LIN {X 0,Y 403.463,Z 460.03,A -85,B 0,C 180,E1 17685.281,E2 17685.281} C_VEL
LIN {X 0,Y 392.488,Z 442.787,A -85,B 0,C 180,E1 17683.008,E2 17683.008} C_VEL
LIN {X 0,Y 381.726,Z 427.301,A -85,B 0,C 180,E1 17680.568,E2 17680.568} C_VEL
LIN {X 0,Y 370.448,Z 412.508,A -85,B 0,C 180,E1 17677.735,E2 17677.735} C_VEL
LIN {X 0,Y 365.323,Z 406.384,A -85,B 0,C 180,E1 17676.338,E2 17676.338} C_VEL
LIN {X 0,Y 362.446,Z 402.418,A -85,B 0,C 180,E1 17675.403,E2 17675.403} C_VEL
LIN {X 0,Y 359.831,Z 397.717,A -85,B 0,C 180,E1 17673.762,E2 17673.762} C_VEL
LIN {X 0,Y 358.471,Z 395.72,A -85,B 0,C 180,E1 17672.95,E2 17672.95} C_VEL
LIN {X 0,Y 356.459,Z 391.629,A -85,B 0,C 180,E1 17671.448,E2 17671.448} C_VEL
LIN {X 0,Y 354.433,Z 388.786,A -85,B 0,C 180,E1 17670.142,E2 17670.142} C_VEL
LIN {X 0,Y 353.887,Z 386.869,A -85,B 0,C 180,E1 17669.398,E2 17669.398} C_VEL
LIN {X 0,Y 353.858,Z 386.651,A -85,B 0,C 180,E1 17665.436,E2 17665.436} C_VEL
LIN {X 0,Y 353.853,Z 386.657,A -85,B 0,C 180,E1 17661.204,E2 17661.204} C_VEL
LIN {X 0,Y 353.849,Z 386.658,A -85,B 0,C 180,E1 17657.09,E2 17657.09} C_VEL
LIN {X 0,Y 353.851,Z 386.655,A -85,B 0,C 180,E1 17653.065,E2 17653.065} C_VEL
LIN {X 0,Y 353.847,Z 386.65,A -85,B 0,C 180,E1 17648.941,E2 17648.941} C_VEL
LIN {X 0,Y 353.843,Z 386.642,A -85,B 0,C 180,E1 17644.863,E2 17644.863} C_VEL
LIN {X 0,Y 353.835,Z 386.641,A -85,B 0,C 180,E1 17640.648,E2 17640.648} C_VEL
LIN {X 0,Y 353.831,Z 386.639,A -85,B 0,C 180,E1 17636.598,E2 17636.598} C_VEL
LIN {X 0,Y 353.837,Z 386.638,A -85,B 0,C 180,E1 17632.532,E2 17632.532} C_VEL
LIN {X 0,Y 353.829,Z 386.639,A -85,B 0,C 180,E1 17628.426,E2 17628.426} C_VEL
LIN {X 0,Y 353.825,Z 386.642,A -85,B 0,C 180,E1 17624.26,E2 17624.26} C_VEL
LIN {X 0,Y 353.839,Z 386.746,A -85,B 0,C 180,E1 17620.523,E2 17620.523} C_VEL
LIN {X 0,Y 354.207,Z 388.34,A -85,B 0,C 180,E1 17619.856,E2 17619.856} C_VEL
LIN {X 0,Y 356.199,Z 391.406,A -85,B 0,C 180,E1 17618.598,E2 17618.598} C_VEL
LIN {X 0,Y 357.309,Z 392.844,A -85,B 0,C 180,E1 17617.978,E2 17617.978} C_VEL
LIN {X 0,Y 359.294,Z 396.484,A -85,B 0,C 180,E1 17616.724,E2 17616.724} C_VEL
LIN {X 0,Y 360.473,Z 398.042,A -85,B 0,C 180,E1 17616.111,E2 17616.111} C_VEL
LIN {X 0,Y 362.61,Z 401.899,A -85,B 0,C 180,E1 17614.873,E2 17614.873} C_VEL
LIN {X 0,Y 363.731,Z 403.854,A -85,B 0,C 180,E1 17614.258,E2 17614.258} C_VEL
LIN {X 0,Y 366.651,Z 408.927,A -85,B 0,C 180,E1 17612.734,E2 17612.734} C_VEL
LIN {X 0,Y 369.981,Z 414.917,A -85,B 0,C 180,E1 17611.07,E2 17611.07} C_VEL
LIN {X 0,Y 374.091,Z 422.477,A -85,B 0,C 180,E1 17609.125,E2 17609.125} C_VEL
LIN {X 0,Y 380.392,Z 434.798,A -85,B 0,C 180,E1 17606.316,E2 17606.316} C_VEL
LIN {X 0,Y 382.59,Z 438.943,A -85,B 0,C 180,E1 17605.52,E2 17605.52} C_VEL
LIN {X 0,Y 392.217,Z 454.061,A -85,B 0,C 180,E1 17603.311,E2 17603.311} C_VEL
LIN {X 0,Y 402.215,Z 471.066,A -85,B 0,C 180,E1 17601.19,E2 17601.19} C_VEL
LIN {X 0,Y 403.176,Z 473.296,A -85,B 0,C 180,E1 17600.98,E2 17600.98} C_VEL
LIN {X 0,Y 405.136,Z 498.631,A -85,B 0,C 180,E1 17600.003,E2 17600.003} C_VEL
LIN {X 0,Y 395.268,Z 723.239,A -85,B 0,C 180,E1 17595.557,E2 17595.557} C_VEL
LIN {X 0,Y 393.737,Z 748.587,A -85,B 0,C 180,E1 17594.972,E2 17594.972} C_VEL
LIN {X 0,Y 391.268,Z 771.267,A -85,B 0,C 180,E1 17594.239,E2 17594.239} C_VEL
LIN {X 0,Y 388.306,Z 792.146,A -85,B 0,C 180,E1 17593.329,E2 17593.329} C_VEL
LIN {X 0,Y 384.904,Z 812.358,A -85,B 0,C 180,E1 17592.178,E2 17592.178} C_VEL
LIN {X 0,Y 380.795,Z 834.172,A -85,B 0,C 180,E1 17590.626,E2 17590.626} C_VEL
LIN {X 0,Y 376.722,Z 854.159,A -85,B 0,C 180,E1 17588.876,E2 17588.876} C_VEL
LIN {X 0,Y 372.707,Z 872.71,A -85,B 0,C 180,E1 17586.924,E2 17586.924} C_VEL
LIN {X 0,Y 368.756,Z 890.411,A -85,B 0,C 180,E1 17584.705,E2 17584.705} C_VEL
LIN {X 0,Y 364.732,Z 908.565,A -85,B 0,C 180,E1 17582.013,E2 17582.013} C_VEL
LIN {X 0,Y 361.461,Z 924.026,A -85,B 0,C 180,E1 17579.312,E2 17579.312} C_VEL
LIN {X 0,Y 358.561,Z 938.566,A -85,B 0,C 180,E1 17576.317,E2 17576.317} C_VEL
LIN {X 0,Y 356.353,Z 950.961,A -85,B 0,C 180,E1 17573.303,E2 17573.303} C_VEL
LIN {X 0,Y 354.62,Z 962.641,A -85,B 0,C 180,E1 17569.946,E2 17569.946} C_VEL
LIN {X 0,Y 353.535,Z 972.315,A -85,B 0,C 180,E1 17566.596,E2 17566.596} C_VEL
LIN {X 0,Y 352.953,Z 979.977,A -85,B 0,C 180,E1 17563.264,E2 17563.264} C_VEL
LIN {X 0,Y 352.727,Z 985.943,A -85,B 0,C 180,E1 17559.957,E2 17559.957} C_VEL
LIN {X 0,Y 352.729,Z 989.818,A -85,B 0,C 180,E1 17557.001,E2 17557.001} C_VEL
LIN {X 0,Y 352.826,Z 992.572,A -85,B 0,C 180,E1 17553.737,E2 17553.737} C_VEL
LIN {X 0,Y 352.867,Z 993.592,A -85,B 0,C 180,E1 17550.812,E2 17550.812} C_VEL
LIN {X 0,Y 352.842,Z 993.283,A -85,B 0,C 180,E1 17547.727,E2 17547.727} C_VEL
LIN {X 0,Y 352.785,Z 991.52,A -85,B 0,C 180,E1 17544.798,E2 17544.798} C_VEL
LIN {X 0,Y 352.717,Z 988.222,A -85,B 0,C 180,E1 17541.616,E2 17541.616} C_VEL
LIN {X 0,Y 352.811,Z 983.168,A -85,B 0,C 180,E1 17538.394,E2 17538.394} C_VEL
LIN {X 0,Y 353.17,Z 976.363,A -85,B 0,C 180,E1 17535.073,E2 17535.073} C_VEL
LIN {X 0,Y 353.949,Z 968.18,A -85,B 0,C 180,E1 17531.899,E2 17531.899} C_VEL
LIN {X 0,Y 355.322,Z 957.64,A -85,B 0,C 180,E1 17528.545,E2 17528.545} C_VEL
LIN {X 0,Y 357.259,Z 945.699,A -85,B 0,C 180,E1 17525.358,E2 17525.358} C_VEL
LIN {X 0,Y 359.753,Z 932.382,A -85,B 0,C 180,E1 17522.349,E2 17522.349} C_VEL
LIN {X 0,Y 362.762,Z 917.65,A -85,B 0,C 180,E1 17519.53,E2 17519.53} C_VEL
LIN {X 0,Y 366.487,Z 900.583,A -85,B 0,C 180,E1 17516.749,E2 17516.749} C_VEL
LIN {X 0,Y 370.396,Z 883.117,A -85,B 0,C 180,E1 17514.338,E2 17514.338} C_VEL
LIN {X 0,Y 374.564,Z 864.11,A -85,B 0,C 180,E1 17512.129,E2 17512.129} C_VEL
LIN {X 0,Y 378.612,Z 844.945,A -85,B 0,C 180,E1 17510.282,E2 17510.282} C_VEL
LIN {X 0,Y 382.706,Z 824.25,A -85,B 0,C 180,E1 17508.631,E2 17508.631} C_VEL
LIN {X 0,Y 386.382,Z 803.737,A -85,B 0,C 180,E1 17507.3,E2 17507.3} C_VEL
LIN {X 0,Y 389.712,Z 782.291,A -85,B 0,C 180,E1 17506.212,E2 17506.212} C_VEL
LIN {X 0,Y 392.534,Z 760.407,A -85,B 0,C 180,E1 17505.386,E2 17505.386} C_VEL
LIN {X 0,Y 394.567,Z 736.575,A -85,B 0,C 180,E1 17504.732,E2 17504.732} C_VEL
LIN {X 0,Y 403.793,Z 527.254,A -85,B 0,C 180,E1 17500.565,E2 17500.565} C_VEL
LIN {X 0,Y 405.03,Z 496.004,A -85,B 0,C 180,E1 17499.928,E2 17499.928} C_VEL
LIN {X 0,Y 402.846,Z 472.338,A -85,B 0,C 180,E1 17498.967,E2 17498.967} C_VEL
LIN {X 0,Y 393.453,Z 456.146,A -85,B 0,C 180,E1 17496.987,E2 17496.987} C_VEL
LIN {X 0,Y 383.635,Z 440.593,A -85,B 0,C 180,E1 17494.758,E2 17494.758} C_VEL
LIN {X 0,Y 381.367,Z 436.803,A -85,B 0,C 180,E1 17494.129,E2 17494.129} C_VEL
LIN {X 0,Y 375.006,Z 424.286,A -85,B 0,C 180,E1 17491.326,E2 17491.326} C_VEL
LIN {X 0,Y 370.225,Z 415.38,A -85,B 0,C 180,E1 17489.086,E2 17489.086} C_VEL
LIN {X 0,Y 368.052,Z 411.439,A -85,B 0,C 180,E1 17488.017,E2 17488.017} C_VEL
LIN {X 0,Y 365.384,Z 406.762,A -85,B 0,C 180,E1 17486.665,E2 17486.665} C_VEL
LIN {X 0,Y 362.852,Z 402.172,A -85,B 0,C 180,E1 17485.284,E2 17485.284} C_VEL
LIN {X 0,Y 360.611,Z 398.471,A -85,B 0,C 180,E1 17484.053,E2 17484.053} C_VEL
LIN {X 0,Y 359.835,Z 397.045,A -85,B 0,C 180,E1 17483.586,E2 17483.586} C_VEL
LIN {X 0,Y 357.627,Z 393.782,A -85,B 0,C 180,E1 17482.348,E2 17482.348} C_VEL
LIN {X 0,Y 356.727,Z 391.855,A -85,B 0,C 180,E1 17481.714,E2 17481.714} C_VEL
LIN {X 0,Y 354.521,Z 389.127,A -85,B 0,C 180,E1 17480.47,E2 17480.47} C_VEL
LIN {X 0,Y 353.863,Z 386.862,A -85,B 0,C 180,E1 17479.648,E2 17479.648} C_VEL
LIN {X 0,Y 353.832,Z 386.64,A -85,B 0,C 180,E1 17475.404,E2 17475.404} C_VEL
LIN {X 0,Y 353.827,Z 386.639,A -85,B 0,C 180,E1 17471.243,E2 17471.243} C_VEL
LIN {X 0,Y 353.837,Z 386.636,A -85,B 0,C 180,E1 17467.142,E2 17467.142} C_VEL
LIN {X 0,Y 353.828,Z 386.637,A -85,B 0,C 180,E1 17462.915,E2 17462.915} C_VEL
LIN {X 0,Y 353.84,Z 386.636,A -85,B 0,C 180,E1 17458.866,E2 17458.866} C_VEL
LIN {X 0,Y 353.834,Z 386.636,A -85,B 0,C 180,E1 17454.649,E2 17454.649} C_VEL
LIN {X 0,Y 353.841,Z 386.64,A -85,B 0,C 180,E1 17450.567,E2 17450.567} C_VEL
LIN {X 0,Y 353.843,Z 386.645,A -85,B 0,C 180,E1 17446.394,E2 17446.394} C_VEL
LIN {X 0,Y 353.842,Z 386.649,A -85,B 0,C 180,E1 17442.206,E2 17442.206} C_VEL
LIN {X 0,Y 353.844,Z 386.648,A -85,B 0,C 180,E1 17438.099,E2 17438.099} C_VEL
LIN {X 0,Y 353.846,Z 386.645,A -85,B 0,C 180,E1 17433.957,E2 17433.957} C_VEL
LIN {X 0,Y 353.899,Z 386.908,A -85,B 0,C 180,E1 17430.421,E2 17430.421} C_VEL
LIN {X 0,Y 355.377,Z 390.465,A -85,B 0,C 180,E1 17429.011,E2 17429.011} C_VEL
LIN {X 0,Y 356.975,Z 392.554,A -85,B 0,C 180,E1 17428.036,E2 17428.036} C_VEL
LIN {X 0,Y 358.87,Z 396.213,A -85,B 0,C 180,E1 17426.694,E2 17426.694} C_VEL
LIN {X 0,Y 359.729,Z 397.399,A -85,B 0,C 180,E1 17426.199,E2 17426.199} C_VEL
LIN {X 0,Y 361.671,Z 401.228,A -85,B 0,C 180,E1 17424.898,E2 17424.898} C_VEL
LIN {X 0,Y 362.955,Z 403.458,A -85,B 0,C 180,E1 17424.218,E2 17424.218} C_VEL
LIN {X 0,Y 367.968,Z 409.61,A -85,B 0,C 180,E1 17422.801,E2 17422.801} C_VEL
LIN {X 0,Y 375.123,Z 418.593,A -85,B 0,C 180,E1 17420.922,E2 17420.922} C_VEL
LIN {X 0,Y 385.584,Z 432.804,A -85,B 0,C 180,E1 17418.407,E2 17418.407} C_VEL
LIN {X 0,Y 396.019,Z 448.184,A -85,B 0,C 180,E1 17416.127,E2 17416.127} C_VEL
LIN {X 0,Y 403.46,Z 460.331,A -85,B 0,C 180,E1 17414.606,E2 17414.606} C_VEL
LIN {X 0,Y 395.816,Z 665.528,A -85,B 0,C 180,E1 17410.809,E2 17410.809} C_VEL
LIN {X 0,Y 394.543,Z 685.835,A -85,B 0,C 180,E1 17410.181,E2 17410.181} C_VEL
LIN {X 0,Y 392.561,Z 706.016,A -85,B 0,C 180,E1 17409.304,E2 17409.304} C_VEL
LIN {X 0,Y 390.075,Z 724.787,A -85,B 0,C 180,E1 17408.24,E2 17408.24} C_VEL
LIN {X 0,Y 386.99,Z 743.305,A -85,B 0,C 180,E1 17406.915,E2 17406.915} C_VEL
LIN {X 0,Y 383.48,Z 760.815,A -85,B 0,C 180,E1 17405.363,E2 17405.363} C_VEL
LIN {X 0,Y 379.684,Z 777.496,A -85,B 0,C 180,E1 17403.57,E2 17403.57} C_VEL
LIN {X 0,Y 375.705,Z 793.271,A -85,B 0,C 180,E1 17401.526,E2 17401.526} C_VEL
LIN {X 0,Y 371.807,Z 807.607,A -85,B 0,C 180,E1 17399.299,E2 17399.299} C_VEL
LIN {X 0,Y 367.752,Z 821.656,A -85,B 0,C 180,E1 17396.651,E2 17396.651} C_VEL
LIN {X 0,Y 364.133,Z 833.715,A -85,B 0,C 180,E1 17393.882,E2 17393.882} C_VEL
LIN {X 0,Y 361.009,Z 844.244,A -85,B 0,C 180,E1 17390.93,E2 17390.93} C_VEL
LIN {X 0,Y 358.326,Z 853.543,A -85,B 0,C 180,E1 17387.705,E2 17387.705} C_VEL
LIN {X 0,Y 356.282,Z 861.241,A -85,B 0,C 180,E1 17384.296,E2 17384.296} C_VEL
LIN {X 0,Y 354.959,Z 866.84,A -85,B 0,C 180,E1 17381.041,E2 17381.041} C_VEL
LIN {X 0,Y 354.134,Z 871.045,A -85,B 0,C 180,E1 17377.624,E2 17377.624} C_VEL
LIN {X 0,Y 353.958,Z 871.872,A -85,B 0,C 180,E1 17376.665,E2 17376.665} C_VEL
LIN {X 0,Y 352.795,Z 873.045,A -85,B 0,C 180,E1 17375.434,E2 17375.434} C_VEL
LIN {X 0,Y 346.257,Z 875.744,A -85,B 0,C 180,E1 17372.045,E2 17372.045} C_VEL
LIN {X 0,Y 345.612,Z 875.991,A -85,B 0,C 180,E1 17371.035,E2 17371.035} C_VEL
LIN {X 0,Y 345.662,Z 875.723,A -85,B 0,C 180,E1 17367.513,E2 17367.513} C_VEL
LIN {X 0,Y 345.969,Z 874.007,A -85,B 0,C 180,E1 17364.028,E2 17364.028} C_VEL
LIN {X 0,Y 346.687,Z 870.505,A -85,B 0,C 180,E1 17360.371,E2 17360.371} C_VEL
LIN {X 0,Y 347.853,Z 865.476,A -85,B 0,C 180,E1 17356.876,E2 17356.876} C_VEL
LIN {X 0,Y 349.613,Z 859.025,A -85,B 0,C 180,E1 17353.554,E2 17353.554} C_VEL
LIN {X 0,Y 352.169,Z 850.32,A -85,B 0,C 180,E1 17350.082,E2 17350.082} C_VEL
LIN {X 0,Y 355.228,Z 840.498,A -85,B 0,C 180,E1 17346.97,E2 17346.97} C_VEL
LIN {X 0,Y 358.578,Z 829.927,A -85,B 0,C 180,E1 17344.218,E2 17344.218} C_VEL
LIN {X 0,Y 362.508,Z 817.205,A -85,B 0,C 180,E1 17341.502,E2 17341.502} C_VEL
LIN {X 0,Y 366.438,Z 803.884,A -85,B 0,C 180,E1 17339.141,E2 17339.141} C_VEL
LIN {X 0,Y 370.835,Z 788.113,A -85,B 0,C 180,E1 17336.819,E2 17336.819} C_VEL
LIN {X 0,Y 374.966,Z 771.814,A -85,B 0,C 180,E1 17334.836,E2 17334.836} C_VEL
LIN {X 0,Y 378.694,Z 755.425,A -85,B 0,C 180,E1 17333.181,E2 17333.181} C_VEL
LIN {X 0,Y 382.2,Z 737.264,A -85,B 0,C 180,E1 17331.687,E2 17331.687} C_VEL
LIN {X 0,Y 385.211,Z 718.333,A -85,B 0,C 180,E1 17330.435,E2 17330.435} C_VEL
LIN {X 0,Y 387.755,Z 697.568,A -85,B 0,C 180,E1 17329.368,E2 17329.368} C_VEL
LIN {X 0,Y 389.51,Z 677.282,A -85,B 0,C 180,E1 17328.604,E2 17328.604} C_VEL
LIN {X 0,Y 390.494,Z 656.885,A -85,B 0,C 180,E1 17328.079,E2 17328.079} C_VEL
LIN {X 0,Y 397.935,Z 463.596,A -85,B 0,C 180,E1 17324.483,E2 17324.483} C_VEL
LIN {X 0,Y 387.854,Z 447.669,A -85,B 0,C 180,E1 17322.312,E2 17322.312} C_VEL
LIN {X 0,Y 377.719,Z 433.028,A -85,B 0,C 180,E1 17319.936,E2 17319.936} C_VEL
LIN {X 0,Y 367.283,Z 419.15,A -85,B 0,C 180,E1 17317.232,E2 17317.232} C_VEL
LIN {X 0,Y 362.237,Z 413.031,A -85,B 0,C 180,E1 17315.815,E2 17315.815} C_VEL
LIN {X 0,Y 358.218,Z 408.108,A -85,B 0,C 180,E1 17314.612,E2 17314.612} C_VEL
LIN {X 0,Y 354.923,Z 403.891,A -85,B 0,C 180,E1 17313.51,E2 17313.51} C_VEL
LIN {X 0,Y 352.123,Z 398.833,A -85,B 0,C 180,E1 17311.594,E2 17311.594} C_VEL
LIN {X 0,Y 349.443,Z 394.421,A -85,B 0,C 180,E1 17309.67,E2 17309.67} C_VEL
LIN {X 0,Y 348.662,Z 392.763,A -85,B 0,C 180,E1 17308.989,E2 17308.989} C_VEL
LIN {X 0,Y 346.325,Z 389.362,A -85,B 0,C 180,E1 17307.236,E2 17307.236} C_VEL
LIN {X 0,Y 345.902,Z 387.676,A -85,B 0,C 180,E1 17306.363,E2 17306.363} C_VEL
LIN {X 0,Y 345.891,Z 387.63,A -85,B 0,C 180,E1 17302.252,E2 17302.252} C_VEL
LIN {X 0,Y 345.894,Z 387.631,A -85,B 0,C 180,E1 17298.017,E2 17298.017} C_VEL
LIN {X 0,Y 345.889,Z 387.631,A -85,B 0,C 180,E1 17293.883,E2 17293.883} C_VEL
LIN {X 0,Y 345.89,Z 387.629,A -85,B 0,C 180,E1 17289.652,E2 17289.652} C_VEL
LIN {X 0,Y 345.881,Z 387.625,A -85,B 0,C 180,E1 17285.641,E2 17285.641} C_VEL
LIN {X 0,Y 345.88,Z 387.625,A -85,B 0,C 180,E1 17281.491,E2 17281.491} C_VEL
LIN {X 0,Y 345.876,Z 387.627,A -85,B 0,C 180,E1 17277.349,E2 17277.349} C_VEL
LIN {X 0,Y 345.875,Z 387.628,A -85,B 0,C 180,E1 17273.194,E2 17273.194} C_VEL
LIN {X 0,Y 345.865,Z 387.631,A -85,B 0,C 180,E1 17269.17,E2 17269.17} C_VEL
LIN {X 0,Y 345.861,Z 387.632,A -85,B 0,C 180,E1 17265.091,E2 17265.091} C_VEL
LIN {X 0,Y 345.884,Z 387.864,A -85,B 0,C 180,E1 17263.291,E2 17263.291} C_VEL
LIN {X 0,Y 347.644,Z 391.765,A -85,B 0,C 180,E1 17261.557,E2 17261.557} C_VEL
LIN {X 0,Y 349.462,Z 393.83,A -85,B 0,C 180,E1 17260.443,E2 17260.443} C_VEL
LIN {X 0,Y 351.179,Z 397.308,A -85,B 0,C 180,E1 17259.152,E2 17259.152} C_VEL
LIN {X 0,Y 352.64,Z 398.867,A -85,B 0,C 180,E1 17258.371,E2 17258.371} C_VEL
LIN {X 0,Y 354.519,Z 402.621,A -85,B 0,C 180,E1 17257.095,E2 17257.095} C_VEL
LIN {X 0,Y 355.964,Z 404.736,A -85,B 0,C 180,E1 17256.293,E2 17256.293} C_VEL
LIN {X 0,Y 358.924,Z 409.885,A -85,B 0,C 180,E1 17254.596,E2 17254.596} C_VEL
LIN {X 0,Y 362.058,Z 415.543,A -85,B 0,C 180,E1 17252.893,E2 17252.893} C_VEL
LIN {X 0,Y 366.595,Z 423.653,A -85,B 0,C 180,E1 17250.598,E2 17250.598} C_VEL
LIN {X 0,Y 373.45,Z 436.875,A -85,B 0,C 180,E1 17247.443,E2 17247.443} C_VEL
LIN {X 0,Y 383.484,Z 452.205,A -85,B 0,C 180,E1 17244.947,E2 17244.947} C_VEL
LIN {X 0,Y 394.336,Z 470.216,A -85,B 0,C 180,E1 17242.494,E2 17242.494} C_VEL
LIN {X 0,Y 397.965,Z 477.117,A -85,B 0,C 180,E1 17241.706,E2 17241.706} C_VEL
LIN {X 0,Y 399.624,Z 499.785,A -85,B 0,C 180,E1 17240.817,E2 17240.817} C_VEL
LIN {X 0,Y 389.299,Z 725.217,A -85,B 0,C 180,E1 17236.312,E2 17236.312} C_VEL
LIN {X 0,Y 387.744,Z 748.686,A -85,B 0,C 180,E1 17235.751,E2 17235.751} C_VEL
LIN {X 0,Y 385.037,Z 772.079,A -85,B 0,C 180,E1 17234.971,E2 17234.971} C_VEL
LIN {X 0,Y 381.897,Z 792.993,A -85,B 0,C 180,E1 17234.032,E2 17234.032} C_VEL
LIN {X 0,Y 378.389,Z 812.868,A -85,B 0,C 180,E1 17232.872,E2 17232.872} C_VEL
LIN {X 0,Y 374.294,Z 833.496,A -85,B 0,C 180,E1 17231.373,E2 17231.373} C_VEL
LIN {X 0,Y 370.062,Z 853.299,A -85,B 0,C 180,E1 17229.612,E2 17229.612} C_VEL
LIN {X 0,Y 365.713,Z 872.448,A -85,B 0,C 180,E1 17227.563,E2 17227.563} C_VEL
LIN {X 0,Y 361.391,Z 890.794,A -85,B 0,C 180,E1 17225.199,E2 17225.199} C_VEL
LIN {X 0,Y 357.383,Z 907.924,A -85,B 0,C 180,E1 17222.583,E2 17222.583} C_VEL
LIN {X 0,Y 353.917,Z 923.361,A -85,B 0,C 180,E1 17219.814,E2 17219.814} C_VEL
LIN {X 0,Y 350.868,Z 937.84,A -85,B 0,C 180,E1 17216.757,E2 17216.757} C_VEL
LIN {X 0,Y 348.439,Z 950.769,A -85,B 0,C 180,E1 17213.505,E2 17213.505} C_VEL
LIN {X 0,Y 346.659,Z 962.235,A -85,B 0,C 180,E1 17210.072,E2 17210.072} C_VEL
LIN {X 0,Y 345.581,Z 971.522,A -85,B 0,C 180,E1 17206.731,E2 17206.731} C_VEL
LIN {X 0,Y 345.005,Z 978.93,A -85,B 0,C 180,E1 17203.405,E2 17203.405} C_VEL
LIN {X 0,Y 344.795,Z 984.818,A -85,B 0,C 180,E1 17200.02,E2 17200.02} C_VEL
LIN {X 0,Y 344.81,Z 988.652,A -85,B 0,C 180,E1 17196.995,E2 17196.995} C_VEL
LIN {X 0,Y 344.933,Z 991.32,A -85,B 0,C 180,E1 17193.657,E2 17193.657} C_VEL
LIN {X 0,Y 344.974,Z 992.289,A -85,B 0,C 180,E1 17190.665,E2 17190.665} C_VEL
LIN {X 0,Y 344.943,Z 991.874,A -85,B 0,C 180,E1 17187.509,E2 17187.509} C_VEL
LIN {X 0,Y 344.873,Z 990.045,A -85,B 0,C 180,E1 17184.511,E2 17184.511} C_VEL
LIN {X 0,Y 344.784,Z 986.492,A -85,B 0,C 180,E1 17181.16,E2 17181.16} C_VEL
LIN {X 0,Y 344.877,Z 981.786,A -85,B 0,C 180,E1 17178.123,E2 17178.123} C_VEL
LIN {X 0,Y 345.285,Z 974.758,A -85,B 0,C 180,E1 17174.639,E2 17174.639} C_VEL
LIN {X 0,Y 346.145,Z 966.289,A -85,B 0,C 180,E1 17171.302,E2 17171.302} C_VEL
LIN {X 0,Y 347.557,Z 956.182,A -85,B 0,C 180,E1 17168.041,E2 17168.041} C_VEL
LIN {X 0,Y 349.629,Z 944.214,A -85,B 0,C 180,E1 17164.783,E2 17164.783} C_VEL
LIN {X 0,Y 352.431,Z 930.272,A -85,B 0,C 180,E1 17161.579,E2 17161.579} C_VEL
LIN {X 0,Y 355.719,Z 915.206,A -85,B 0,C 180,E1 17158.672,E2 17158.672} C_VEL
LIN {X 0,Y 359.476,Z 898.845,A -85,B 0,C 180,E1 17155.982,E2 17155.982} C_VEL
LIN {X 0,Y 363.577,Z 881.519,A -85,B 0,C 180,E1 17153.563,E2 17153.563} C_VEL
LIN {X 0,Y 367.964,Z 862.494,A -85,B 0,C 180,E1 17151.325,E2 17151.325} C_VEL
LIN {X 0,Y 372.235,Z 843.272,A -85,B 0,C 180,E1 17149.461,E2 17149.461} C_VEL
LIN {X 0,Y 376.507,Z 822.479,A -85,B 0,C 180,E1 17147.794,E2 17147.794} C_VEL
LIN {X 0,Y 380.409,Z 801.412,A -85,B 0,C 180,E1 17146.432,E2 17146.432} C_VEL
LIN {X 0,Y 383.965,Z 779.517,A -85,B 0,C 180,E1 17145.331,E2 17145.331} C_VEL
LIN {X 0,Y 386.835,Z 757.431,A -85,B 0,C 180,E1 17144.516,E2 17144.516} C_VEL
LIN {X 0,Y 388.75,Z 734.671,A -85,B 0,C 180,E1 17143.9,E2 17143.9} C_VEL
LIN {X 0,Y 398.548,Z 521.369,A -85,B 0,C 180,E1 17139.617,E2 17139.617} C_VEL
LIN {X 0,Y 399.513,Z 497.254,A -85,B 0,C 180,E1 17139.115,E2 17139.115} C_VEL
LIN {X 0,Y 397.675,Z 476.357,A -85,B 0,C 180,E1 17138.253,E2 17138.253} C_VEL
LIN {X 0,Y 387.152,Z 458.169,A -85,B 0,C 180,E1 17135.937,E2 17135.937} C_VEL
LIN {X 0,Y 376.915,Z 442.175,A -85,B 0,C 180,E1 17133.488,E2 17133.488} C_VEL
LIN {X 0,Y 372.86,Z 435.795,A -85,B 0,C 180,E1 17132.37,E2 17132.37} C_VEL
LIN {X 0,Y 365.961,Z 422.45,A -85,B 0,C 180,E1 17129.099,E2 17129.099} C_VEL
LIN {X 0,Y 360.529,Z 412.822,A -85,B 0,C 180,E1 17126.342,E2 17126.342} C_VEL
LIN {X 0,Y 358.01,Z 408.293,A -85,B 0,C 180,E1 17124.943,E2 17124.943} C_VEL
LIN {X 0,Y 355.032,Z 403.224,A -85,B 0,C 180,E1 17123.22,E2 17123.22} C_VEL
LIN {X 0,Y 352.75,Z 399.261,A -85,B 0,C 180,E1 17121.796,E2 17121.796} C_VEL
LIN {X 0,Y 349.91,Z 395.168,A -85,B 0,C 180,E1 17120.053,E2 17120.053} C_VEL
LIN {X 0,Y 349.196,Z 393.201,A -85,B 0,C 180,E1 17119.399,E2 17119.399} C_VEL
LIN {X 0,Y 346.669,Z 390.23,A -85,B 0,C 180,E1 17117.801,E2 17117.801} C_VEL
LIN {X 0,Y 345.891,Z 387.897,A -85,B 0,C 180,E1 17116.802,E2 17116.802} C_VEL
LIN {X 0,Y 345.885,Z 387.652,A -85,B 0,C 180,E1 17113.201,E2 17113.201} C_VEL
LIN {X 0,Y 345.88,Z 387.65,A -85,B 0,C 180,E1 17108.98,E2 17108.98} C_VEL
LIN {X 0,Y 345.881,Z 387.651,A -85,B 0,C 180,E1 17104.808,E2 17104.808} C_VEL
LIN {X 0,Y 345.883,Z 387.653,A -85,B 0,C 180,E1 17100.662,E2 17100.662} C_VEL
LIN {X 0,Y 345.883,Z 387.645,A -85,B 0,C 180,E1 17096.519,E2 17096.519} C_VEL
LIN {X 0,Y 345.884,Z 387.637,A -85,B 0,C 180,E1 17092.358,E2 17092.358} C_VEL
LIN {X 0,Y 345.883,Z 387.635,A -85,B 0,C 180,E1 17088.156,E2 17088.156} C_VEL
LIN {X 0,Y 345.889,Z 387.633,A -85,B 0,C 180,E1 17084.06,E2 17084.06} C_VEL
LIN {X 0,Y 345.89,Z 387.633,A -85,B 0,C 180,E1 17079.879,E2 17079.879} C_VEL
LIN {X 0,Y 345.893,Z 387.634,A -85,B 0,C 180,E1 17075.765,E2 17075.765} C_VEL
LIN {X 0,Y 345.922,Z 387.883,A -85,B 0,C 180,E1 17073.257,E2 17073.257} C_VEL
LIN {X 0,Y 347.896,Z 392.024,A -85,B 0,C 180,E1 17071.317,E2 17071.317} C_VEL
LIN {X 0,Y 349.163,Z 393.487,A -85,B 0,C 180,E1 17070.492,E2 17070.492} C_VEL
LIN {X 0,Y 350.909,Z 397.141,A -85,B 0,C 180,E1 17069.043,E2 17069.043} C_VEL
LIN {X 0,Y 352.092,Z 398.707,A -85,B 0,C 180,E1 17068.307,E2 17068.307} C_VEL
LIN {X 0,Y 353.924,Z 402.337,A -85,B 0,C 180,E1 17066.959,E2 17066.959} C_VEL
LIN {X 0,Y 355.083,Z 404.243,A -85,B 0,C 180,E1 17066.26,E2 17066.26} C_VEL
LIN {X 0,Y 358.728,Z 408.57,A -85,B 0,C 180,E1 17065.104,E2 17065.104} C_VEL
LIN {X 0,Y 365.33,Z 416.873,A -85,B 0,C 180,E1 17063.175,E2 17063.175} C_VEL
LIN {X 0,Y 372.147,Z 425.547,A -85,B 0,C 180,E1 17061.342,E2 17061.342} C_VEL
LIN {X 0,Y 382.216,Z 439.434,A -85,B 0,C 180,E1 17058.859,E2 17058.859} C_VEL
LIN {X 0,Y 392.243,Z 454.456,A -85,B 0,C 180,E1 17056.608,E2 17056.608} C_VEL
LIN {X 0,Y 397.974,Z 463.927,A -85,B 0,C 180,E1 17055.395,E2 17055.395} C_VEL
LIN {X 0,Y 390.052,Z 666.386,A -85,B 0,C 180,E1 17051.609,E2 17051.609} C_VEL
LIN {X 0,Y 388.73,Z 686.692,A -85,B 0,C 180,E1 17050.975,E2 17050.975} C_VEL
LIN {X 0,Y 386.644,Z 707.132,A -85,B 0,C 180,E1 17050.079,E2 17050.079} C_VEL
LIN {X 0,Y 384.144,Z 725.404,A -85,B 0,C 180,E1 17049.036,E2 17049.036} C_VEL
LIN {X 0,Y 380.928,Z 743.984,A -85,B 0,C 180,E1 17047.699,E2 17047.699} C_VEL
LIN {X 0,Y 377.244,Z 761.731,A -85,B 0,C 180,E1 17046.115,E2 17046.115} C_VEL
LIN {X 0,Y 373.316,Z 778.349,A -85,B 0,C 180,E1 17044.313,E2 17044.313} C_VEL
LIN {X 0,Y 369.162,Z 794.191,A -85,B 0,C 180,E1 17042.242,E2 17042.242} C_VEL
LIN {X 0,Y 364.94,Z 809.02,A -85,B 0,C 180,E1 17039.906,E2 17039.906} C_VEL
LIN {X 0,Y 360.927,Z 822.274,A -85,B 0,C 180,E1 17037.375,E2 17037.375} C_VEL
LIN {X 0,Y 357.204,Z 834.106,A -85,B 0,C 180,E1 17034.646,E2 17034.646} C_VEL
LIN {X 0,Y 353.841,Z 844.887,A -85,B 0,C 180,E1 17031.616,E2 17031.616} C_VEL
LIN {X 0,Y 351.027,Z 854.072,A -85,B 0,C 180,E1 17028.429,E2 17028.429} C_VEL
LIN {X 0,Y 348.885,Z 861.641,A -85,B 0,C 180,E1 17025.115,E2 17025.115} C_VEL
LIN {X 0,Y 347.308,Z 867.731,A -85,B 0,C 180,E1 17021.624,E2 17021.624} C_VEL
LIN {X 0,Y 346.323,Z 872.204,A -85,B 0,C 180,E1 17017.964,E2 17017.964} C_VEL
LIN {X 0,Y 345.803,Z 874.838,A -85,B 0,C 180,E1 17014.477,E2 17014.477} C_VEL
LIN {X 0,Y 345.612,Z 875.991,A -85,B 0,C 180,E1 17011.035,E2 17011.035} C_VEL
LIN {X 0,Y 344.636,Z 876.264,A -85,B 0,C 180,E1 17009.758,E2 17009.758} C_VEL
LIN {X 0,Y 338.487,Z 876.549,A -85,B 0,C 180,E1 17006.238,E2 17006.238} C_VEL
LIN {X 0,Y 337.943,Z 876.107,A -85,B 0,C 180,E1 17005.205,E2 17005.205} C_VEL
LIN {X 0,Y 338.506,Z 873.471,A -85,B 0,C 180,E1 17001.678,E2 17001.678} C_VEL
LIN {X 0,Y 339.519,Z 869.207,A -85,B 0,C 180,E1 16998.104,E2 16998.104} C_VEL
LIN {X 0,Y 341.186,Z 863.175,A -85,B 0,C 180,E1 16994.534,E2 16994.534} C_VEL
LIN {X 0,Y 343.445,Z 855.671,A -85,B 0,C 180,E1 16991.148,E2 16991.148} C_VEL
LIN {X 0,Y 346.504,Z 846.234,A -85,B 0,C 180,E1 16987.791,E2 16987.791} C_VEL
LIN {X 0,Y 350.137,Z 835.206,A -85,B 0,C 180,E1 16984.64,E2 16984.64} C_VEL
LIN {X 0,Y 354.06,Z 823.328,A -85,B 0,C 180,E1 16981.864,E2 16981.864} C_VEL
LIN {X 0,Y 358.369,Z 809.758,A -85,B 0,C 180,E1 16979.242,E2 16979.242} C_VEL
LIN {X 0,Y 362.866,Z 794.635,A -85,B 0,C 180,E1 16976.845,E2 16976.845} C_VEL
LIN {X 0,Y 367.106,Z 779.018,A -85,B 0,C 180,E1 16974.795,E2 16974.795} C_VEL
LIN {X 0,Y 371.347,Z 761.641,A -85,B 0,C 180,E1 16972.91,E2 16972.91} C_VEL
LIN {X 0,Y 375.074,Z 744.207,A -85,B 0,C 180,E1 16971.359,E2 16971.359} C_VEL
LIN {X 0,Y 378.4,Z 725.683,A -85,B 0,C 180,E1 16970.021,E2 16970.021} C_VEL
LIN {X 0,Y 381.117,Z 706.206,A -85,B 0,C 180,E1 16968.919,E2 16968.919} C_VEL
LIN {X 0,Y 383.161,Z 686.203,A -85,B 0,C 180,E1 16968.058,E2 16968.058} C_VEL
LIN {X 0,Y 384.533,Z 664.551,A -85,B 0,C 180,E1 16967.406,E2 16967.406} C_VEL
LIN {X 0,Y 392.534,Z 467.167,A -85,B 0,C 180,E1 16963.669,E2 16963.669} C_VEL
LIN {X 0,Y 381.914,Z 450.442,A -85,B 0,C 180,E1 16961.281,E2 16961.281} C_VEL
LIN {X 0,Y 371.579,Z 435.636,A -85,B 0,C 180,E1 16958.728,E2 16958.728} C_VEL
LIN {X 0,Y 363.157,Z 424.624,A -85,B 0,C 180,E1 16956.443,E2 16956.443} C_VEL
LIN {X 0,Y 359.422,Z 419.937,A -85,B 0,C 180,E1 16955.354,E2 16955.354} C_VEL
LIN {X 0,Y 355.457,Z 415.04,A -85,B 0,C 180,E1 16954.137,E2 16954.137} C_VEL
LIN {X 0,Y 350.981,Z 409.643,A -85,B 0,C 180,E1 16952.673,E2 16952.673} C_VEL
LIN {X 0,Y 347.428,Z 405.29,A -85,B 0,C 180,E1 16951.393,E2 16951.393} C_VEL
LIN {X 0,Y 344.634,Z 400.535,A -85,B 0,C 180,E1 16949.361,E2 16949.361} C_VEL
LIN {X 0,Y 344.077,Z 399.279,A -85,B 0,C 180,E1 16948.841,E2 16948.841} C_VEL
LIN {X 0,Y 341.698,Z 395.697,A -85,B 0,C 180,E1 16946.972,E2 16946.972} C_VEL
LIN {X 0,Y 340.848,Z 393.835,A -85,B 0,C 180,E1 16946.105,E2 16946.105} C_VEL
LIN {X 0,Y 338.466,Z 390.58,A -85,B 0,C 180,E1 16944.059,E2 16944.059} C_VEL
LIN {X 0,Y 337.973,Z 388.727,A -85,B 0,C 180,E1 16942.987,E2 16942.987} C_VEL
LIN {X 0,Y 337.953,Z 388.613,A -85,B 0,C 180,E1 16938.798,E2 16938.798} C_VEL
LIN {X 0,Y 337.943,Z 388.615,A -85,B 0,C 180,E1 16934.566,E2 16934.566} C_VEL
LIN {X 0,Y 337.94,Z 388.614,A -85,B 0,C 180,E1 16930.398,E2 16930.398} C_VEL
LIN {X 0,Y 337.933,Z 388.614,A -85,B 0,C 180,E1 16926.115,E2 16926.115} C_VEL
LIN {X 0,Y 337.93,Z 388.615,A -85,B 0,C 180,E1 16921.866,E2 16921.866} C_VEL
LIN {X 0,Y 337.928,Z 388.617,A -85,B 0,C 180,E1 16917.626,E2 16917.626} C_VEL
LIN {X 0,Y 337.929,Z 388.618,A -85,B 0,C 180,E1 16913.374,E2 16913.374} C_VEL
LIN {X 0,Y 337.926,Z 388.619,A -85,B 0,C 180,E1 16909.184,E2 16909.184} C_VEL
LIN {X 0,Y 337.996,Z 388.915,A -85,B 0,C 180,E1 16906.66,E2 16906.66} C_VEL
LIN {X 0,Y 339.524,Z 392.492,A -85,B 0,C 180,E1 16904.806,E2 16904.806} C_VEL
LIN {X 0,Y 341.589,Z 394.746,A -85,B 0,C 180,E1 16903.331,E2 16903.331} C_VEL
LIN {X 0,Y 343.514,Z 398.581,A -85,B 0,C 180,E1 16901.679,E2 16901.679} C_VEL
LIN {X 0,Y 345.048,Z 400.381,A -85,B 0,C 180,E1 16900.711,E2 16900.711} C_VEL
LIN {X 0,Y 347.031,Z 404.143,A -85,B 0,C 180,E1 16899.245,E2 16899.245} C_VEL
LIN {X 0,Y 348.156,Z 405.458,A -85,B 0,C 180,E1 16898.61,E2 16898.61} C_VEL
LIN {X 0,Y 350.34,Z 409.477,A -85,B 0,C 180,E1 16897.162,E2 16897.162} C_VEL
LIN {X 0,Y 351.408,Z 411.229,A -85,B 0,C 180,E1 16896.526,E2 16896.526} C_VEL
LIN {X 0,Y 354.363,Z 416.483,A -85,B 0,C 180,E1 16894.783,E2 16894.783} C_VEL
LIN {X 0,Y 357.403,Z 422.077,A -85,B 0,C 180,E1 16893.051,E2 16893.051} C_VEL
LIN {X 0,Y 361.734,Z 429.845,A -85,B 0,C 180,E1 16890.852,E2 16890.852} C_VEL
LIN {X 0,Y 365.161,Z 436.29,A -85,B 0,C 180,E1 16889.293,E2 16889.293} C_VEL
LIN {X 0,Y 374.606,Z 450.198,A -85,B 0,C 180,E1 16886.759,E2 16886.759} C_VEL
LIN {X 0,Y 384.459,Z 466.195,A -85,B 0,C 180,E1 16884.347,E2 16884.347} C_VEL
LIN {X 0,Y 392.804,Z 480.84,A -85,B 0,C 180,E1 16882.455,E2 16882.455} C_VEL
LIN {X 0,Y 394.186,Z 501.143,A -85,B 0,C 180,E1 16881.649,E2 16881.649} C_VEL
LIN {X 0,Y 383.404,Z 727.146,A -85,B 0,C 180,E1 16877.092,E2 16877.092} C_VEL
LIN {X 0,Y 381.711,Z 750.09,A -85,B 0,C 180,E1 16876.518,E2 16876.518} C_VEL
LIN {X 0,Y 378.976,Z 772.159,A -85,B 0,C 180,E1 16875.757,E2 16875.757} C_VEL
LIN {X 0,Y 375.55,Z 793.736,A -85,B 0,C 180,E1 16874.76,E2 16874.76} C_VEL
LIN {X 0,Y 371.883,Z 813.64,A -85,B 0,C 180,E1 16873.573,E2 16873.573} C_VEL
LIN {X 0,Y 367.63,Z 833.916,A -85,B 0,C 180,E1 16872.057,E2 16872.057} C_VEL
LIN {X 0,Y 363.095,Z 853.994,A -85,B 0,C 180,E1 16870.217,E2 16870.217} C_VEL
LIN {X 0,Y 358.649,Z 872.594,A -85,B 0,C 180,E1 16868.171,E2 16868.171} C_VEL
LIN {X 0,Y 354.133,Z 890.845,A -85,B 0,C 180,E1 16865.76,E2 16865.76} C_VEL
LIN {X 0,Y 350.111,Z 907.142,A -85,B 0,C 180,E1 16863.201,E2 16863.201} C_VEL
LIN {X 0,Y 346.201,Z 923.547,A -85,B 0,C 180,E1 16860.165,E2 16860.165} C_VEL
LIN {X 0,Y 343.039,Z 937.814,A -85,B 0,C 180,E1 16857.043,E2 16857.043} C_VEL
LIN {X 0,Y 340.529,Z 950.583,A -85,B 0,C 180,E1 16853.717,E2 16853.717} C_VEL
LIN {X 0,Y 338.773,Z 961.316,A -85,B 0,C 180,E1 16850.38,E2 16850.38} C_VEL
LIN {X 0,Y 337.626,Z 970.722,A -85,B 0,C 180,E1 16846.87,E2 16846.87} C_VEL
LIN {X 0,Y 337.056,Z 977.887,A -85,B 0,C 180,E1 16843.552,E2 16843.552} C_VEL
LIN {X 0,Y 336.862,Z 983.694,A -85,B 0,C 180,E1 16840.085,E2 16840.085} C_VEL
LIN {X 0,Y 336.892,Z 987.488,A -85,B 0,C 180,E1 16836.989,E2 16836.989} C_VEL
LIN {X 0,Y 337.031,Z 989.985,A -85,B 0,C 180,E1 16833.742,E2 16833.742} C_VEL
LIN {X 0,Y 337.089,Z 990.936,A -85,B 0,C 180,E1 16830.85,E2 16830.85} C_VEL
LIN {X 0,Y 337.051,Z 990.62,A -85,B 0,C 180,E1 16827.621,E2 16827.621} C_VEL
LIN {X 0,Y 336.969,Z 988.838,A -85,B 0,C 180,E1 16824.553,E2 16824.553} C_VEL
LIN {X 0,Y 336.855,Z 985.565,A -85,B 0,C 180,E1 16821.268,E2 16821.268} C_VEL
LIN {X 0,Y 336.929,Z 980.7,A -85,B 0,C 180,E1 16818.013,E2 16818.013} C_VEL
LIN {X 0,Y 337.327,Z 973.952,A -85,B 0,C 180,E1 16814.53,E2 16814.53} C_VEL
LIN {X 0,Y 338.213,Z 965.48,A -85,B 0,C 180,E1 16811.086,E2 16811.086} C_VEL
LIN {X 0,Y 339.71,Z 955.305,A -85,B 0,C 180,E1 16807.689,E2 16807.689} C_VEL
LIN {X 0,Y 341.891,Z 943.436,A -85,B 0,C 180,E1 16804.356,E2 16804.356} C_VEL
LIN {X 0,Y 344.783,Z 929.797,A -85,B 0,C 180,E1 16801.137,E2 16801.137} C_VEL
LIN {X 0,Y 348.293,Z 914.606,A -85,B 0,C 180,E1 16798.119,E2 16798.119} C_VEL
LIN {X 0,Y 352.462,Z 897.474,A -85,B 0,C 180,E1 16795.241,E2 16795.241} C_VEL
LIN {X 0,Y 356.826,Z 879.93,A -85,B 0,C 180,E1 16792.758,E2 16792.758} C_VEL
LIN {X 0,Y 361.377,Z 861.186,A -85,B 0,C 180,E1 16790.528,E2 16790.528} C_VEL
LIN {X 0,Y 365.931,Z 841.605,A -85,B 0,C 180,E1 16788.612,E2 16788.612} C_VEL
LIN {X 0,Y 370.184,Z 821.76,A -85,B 0,C 180,E1 16787.006,E2 16787.006} C_VEL
LIN {X 0,Y 374.134,Z 801.481,A -85,B 0,C 180,E1 16785.672,E2 16785.672} C_VEL
LIN {X 0,Y 377.82,Z 779.695,A -85,B 0,C 180,E1 16784.559,E2 16784.559} C_VEL
LIN {X 0,Y 380.804,Z 757.949,A -85,B 0,C 180,E1 16783.735,E2 16783.735} C_VEL
LIN {X 0,Y 382.923,Z 734.361,A -85,B 0,C 180,E1 16783.078,E2 16783.078} C_VEL
LIN {X 0,Y 392.995,Z 524.135,A -85,B 0,C 180,E1 16778.816,E2 16778.816} C_VEL
LIN {X 0,Y 394.08,Z 498.517,A -85,B 0,C 180,E1 16778.28,E2 16778.28} C_VEL
LIN {X 0,Y 392.565,Z 480.413,A -85,B 0,C 180,E1 16777.52,E2 16777.52} C_VEL
LIN {X 0,Y 382.629,Z 463.115,A -85,B 0,C 180,E1 16775.252,E2 16775.252} C_VEL
LIN {X 0,Y 371.507,Z 445.587,A -85,B 0,C 180,E1 16772.474,E2 16772.474} C_VEL
LIN {X 0,Y 364.074,Z 434.495,A -85,B 0,C 180,E1 16770.352,E2 16770.352} C_VEL
LIN {X 0,Y 358.935,Z 424.5,A -85,B 0,C 180,E1 16767.723,E2 16767.723} C_VEL
LIN {X 0,Y 353.193,Z 414.39,A -85,B 0,C 180,E1 16764.591,E2 16764.591} C_VEL
LIN {X 0,Y 350.55,Z 409.72,A -85,B 0,C 180,E1 16763.001,E2 16763.001} C_VEL
LIN {X 0,Y 348.244,Z 405.758,A -85,B 0,C 180,E1 16761.542,E2 16761.542} C_VEL
LIN {X 0,Y 345.315,Z 401.199,A -85,B 0,C 180,E1 16759.625,E2 16759.625} C_VEL
LIN {X 0,Y 344.765,Z 399.785,A -85,B 0,C 180,E1 16759.13,E2 16759.13} C_VEL
LIN {X 0,Y 342.321,Z 396.71,A -85,B 0,C 180,E1 16757.508,E2 16757.508} C_VEL
LIN {X 0,Y 341.034,Z 394.04,A -85,B 0,C 180,E1 16756.347,E2 16756.347} C_VEL
LIN {X 0,Y 338.505,Z 390.807,A -85,B 0,C 180,E1 16754.366,E2 16754.366} C_VEL
LIN {X 0,Y 337.979,Z 388.815,A -85,B 0,C 180,E1 16753.341,E2 16753.341} C_VEL
LIN {X 0,Y 337.953,Z 388.64,A -85,B 0,C 180,E1 16749.193,E2 16749.193} C_VEL
LIN {X 0,Y 337.949,Z 388.641,A -85,B 0,C 180,E1 16744.922,E2 16744.922} C_VEL
LIN {X 0,Y 337.945,Z 388.641,A -85,B 0,C 180,E1 16740.678,E2 16740.678} C_VEL
LIN {X 0,Y 337.94,Z 388.635,A -85,B 0,C 180,E1 16736.437,E2 16736.437} C_VEL
LIN {X 0,Y 337.938,Z 388.63,A -85,B 0,C 180,E1 16732.177,E2 16732.177} C_VEL
LIN {X 0,Y 337.938,Z 388.629,A -85,B 0,C 180,E1 16727.873,E2 16727.873} C_VEL
LIN {X 0,Y 337.94,Z 388.632,A -85,B 0,C 180,E1 16723.499,E2 16723.499} C_VEL
LIN {X 0,Y 337.949,Z 388.633,A -85,B 0,C 180,E1 16719.198,E2 16719.198} C_VEL
LIN {X 0,Y 338.012,Z 388.885,A -85,B 0,C 180,E1 16716.648,E2 16716.648} C_VEL
LIN {X 0,Y 339.705,Z 392.687,A -85,B 0,C 180,E1 16714.55,E2 16714.55} C_VEL
LIN {X 0,Y 341.349,Z 394.615,A -85,B 0,C 180,E1 16713.289,E2 16713.289} C_VEL
LIN {X 0,Y 343.338,Z 398.534,A -85,B 0,C 180,E1 16711.471,E2 16711.471} C_VEL
LIN {X 0,Y 344.378,Z 399.63,A -85,B 0,C 180,E1 16710.806,E2 16710.806} C_VEL
LIN {X 0,Y 346.188,Z 403.482,A -85,B 0,C 180,E1 16709.255,E2 16709.255} C_VEL
LIN {X 0,Y 347.279,Z 404.885,A -85,B 0,C 180,E1 16708.592,E2 16708.592} C_VEL
LIN {X 0,Y 350.319,Z 409.035,A -85,B 0,C 180,E1 16707.403,E2 16707.403} C_VEL
LIN {X 0,Y 352.543,Z 411.492,A -85,B 0,C 180,E1 16706.667,E2 16706.667} C_VEL
LIN {X 0,Y 357.687,Z 417.808,A -85,B 0,C 180,E1 16705.037,E2 16705.037} C_VEL
LIN {X 0,Y 362.305,Z 423.577,A -85,B 0,C 180,E1 16703.67,E2 16703.67} C_VEL
LIN {X 0,Y 369.189,Z 432.516,A -85,B 0,C 180,E1 16701.768,E2 16701.768} C_VEL
LIN {X 0,Y 378.74,Z 445.863,A -85,B 0,C 180,E1 16699.352,E2 16699.352} C_VEL
LIN {X 0,Y 388.636,Z 460.949,A -85,B 0,C 180,E1 16697.067,E2 16697.067} C_VEL
LIN {X 0,Y 392.566,Z 467.535,A -85,B 0,C 180,E1 16696.206,E2 16696.206} C_VEL
LIN {X 0,Y 384.365,Z 667.231,A -85,B 0,C 180,E1 16692.433,E2 16692.433} C_VEL
LIN {X 0,Y 382.995,Z 687.539,A -85,B 0,C 180,E1 16691.794,E2 16691.794} C_VEL
LIN {X 0,Y 380.865,Z 707.734,A -85,B 0,C 180,E1 16690.904,E2 16690.904} C_VEL
LIN {X 0,Y 378.29,Z 726.014,A -85,B 0,C 180,E1 16689.857,E2 16689.857} C_VEL
LIN {X 0,Y 374.939,Z 744.656,A -85,B 0,C 180,E1 16688.507,E2 16688.507} C_VEL
LIN {X 0,Y 371.137,Z 762.362,A -85,B 0,C 180,E1 16686.92,E2 16686.92} C_VEL
LIN {X 0,Y 366.846,Z 779.834,A -85,B 0,C 180,E1 16685.006,E2 16685.006} C_VEL
LIN {X 0,Y 362.521,Z 795.632,A -85,B 0,C 180,E1 16682.907,E2 16682.907} C_VEL
LIN {X 0,Y 358.395,Z 809.54,A -85,B 0,C 180,E1 16680.696,E2 16680.696} C_VEL
LIN {X 0,Y 354.164,Z 822.887,A -85,B 0,C 180,E1 16678.126,E2 16678.126} C_VEL
LIN {X 0,Y 350.23,Z 834.84,A -85,B 0,C 180,E1 16675.352,E2 16675.352} C_VEL
LIN {X 0,Y 346.529,Z 846.098,A -85,B 0,C 180,E1 16672.149,E2 16672.149} C_VEL
LIN {X 0,Y 343.505,Z 855.429,A -85,B 0,C 180,E1 16668.848,E2 16668.848} C_VEL
LIN {X 0,Y 341.233,Z 862.989,A -85,B 0,C 180,E1 16665.462,E2 16665.462} C_VEL
LIN {X 0,Y 339.548,Z 869.073,A -85,B 0,C 180,E1 16661.894,E2 16661.894} C_VEL
LIN {X 0,Y 338.523,Z 873.359,A -85,B 0,C 180,E1 16658.32,E2 16658.32} C_VEL
LIN {X 0,Y 337.947,Z 876.07,A -85,B 0,C 180,E1 16654.751,E2 16654.751} C_VEL
LIN {X 0,Y 337.724,Z 877.324,A -85,B 0,C 180,E1 16651.017,E2 16651.017} C_VEL
LIN {X 0,Y 337.777,Z 877.052,A -85,B 0,C 180,E1 16647.455,E2 16647.455} C_VEL
LIN {X 0,Y 337.943,Z 876.107,A -85,B 0,C 180,E1 16645.205,E2 16645.205} C_VEL
LIN {X 0,Y 337.126,Z 875.525,A -85,B 0,C 180,E1 16643.899,E2 16643.899} C_VEL
LIN {X 0,Y 331.614,Z 873.504,A -85,B 0,C 180,E1 16640.291,E2 16640.291} C_VEL
LIN {X 0,Y 331.265,Z 872.383,A -85,B 0,C 180,E1 16639.251,E2 16639.251} C_VEL
LIN {X 0,Y 332.775,Z 867.048,A -85,B 0,C 180,E1 16635.56,E2 16635.56} C_VEL
LIN {X 0,Y 335.02,Z 859.905,A -85,B 0,C 180,E1 16631.919,E2 16631.919} C_VEL
LIN {X 0,Y 337.952,Z 851.162,A -85,B 0,C 180,E1 16628.479,E2 16628.479} C_VEL
LIN {X 0,Y 341.287,Z 841.486,A -85,B 0,C 180,E1 16625.419,E2 16625.419} C_VEL
LIN {X 0,Y 345.429,Z 829.565,A -85,B 0,C 180,E1 16622.342,E2 16622.342} C_VEL
LIN {X 0,Y 349.78,Z 816.654,A -85,B 0,C 180,E1 16619.608,E2 16619.608} C_VEL
LIN {X 0,Y 354.24,Z 802.879,A -85,B 0,C 180,E1 16617.188,E2 16617.188} C_VEL
LIN {X 0,Y 358.849,Z 787.241,A -85,B 0,C 180,E1 16614.923,E2 16614.923} C_VEL
LIN {X 0,Y 363.121,Z 771.304,A -85,B 0,C 180,E1 16613.016,E2 16613.016} C_VEL
LIN {X 0,Y 367.364,Z 753.406,A -85,B 0,C 180,E1 16611.249,E2 16611.249} C_VEL
LIN {X 0,Y 370.99,Z 735.465,A -85,B 0,C 180,E1 16609.803,E2 16609.803} C_VEL
LIN {X 0,Y 374.203,Z 716.025,A -85,B 0,C 180,E1 16608.553,E2 16608.553} C_VEL
LIN {X 0,Y 376.668,Z 696.083,A -85,B 0,C 180,E1 16607.572,E2 16607.572} C_VEL
LIN {X 0,Y 378.367,Z 676.102,A -85,B 0,C 180,E1 16606.849,E2 16606.849} C_VEL
LIN {X 0,Y 379.456,Z 652.227,A -85,B 0,C 180,E1 16606.274,E2 16606.274} C_VEL
LIN {X 0,Y 387.231,Z 470.892,A -85,B 0,C 180,E1 16602.841,E2 16602.841} C_VEL
LIN {X 0,Y 376.938,Z 454.593,A -85,B 0,C 180,E1 16600.428,E2 16600.428} C_VEL
LIN {X 0,Y 367.467,Z 441.091,A -85,B 0,C 180,E1 16597.997,E2 16597.997} C_VEL
LIN {X 0,Y 359.949,Z 431.073,A -85,B 0,C 180,E1 16595.882,E2 16595.882} C_VEL
LIN {X 0,Y 353.07,Z 422.32,A -85,B 0,C 180,E1 16593.763,E2 16593.763} C_VEL
LIN {X 0,Y 348.208,Z 416.508,A -85,B 0,C 180,E1 16592.137,E2 16592.137} C_VEL
LIN {X 0,Y 343.704,Z 411.165,A -85,B 0,C 180,E1 16590.507,E2 16590.507} C_VEL
LIN {X 0,Y 340.082,Z 406.889,A -85,B 0,C 180,E1 16589.068,E2 16589.068} C_VEL
LIN {X 0,Y 339.299,Z 405.578,A -85,B 0,C 180,E1 16588.515,E2 16588.515} C_VEL
LIN {X 0,Y 337.009,Z 401.83,A -85,B 0,C 180,E1 16586.616,E2 16586.616} C_VEL
LIN {X 0,Y 336.332,Z 400.384,A -85,B 0,C 180,E1 16585.913,E2 16585.913} C_VEL
LIN {X 0,Y 334.032,Z 397.117,A -85,B 0,C 180,E1 16583.835,E2 16583.835} C_VEL
LIN {X 0,Y 333.226,Z 395.097,A -85,B 0,C 180,E1 16582.773,E2 16582.773} C_VEL
LIN {X 0,Y 330.571,Z 391.683,A -85,B 0,C 180,E1 16579.986,E2 16579.986} C_VEL
LIN {X 0,Y 330.051,Z 389.878,A -85,B 0,C 180,E1 16578.731,E2 16578.731} C_VEL
LIN {X 0,Y 330.012,Z 389.601,A -85,B 0,C 180,E1 16574.744,E2 16574.744} C_VEL
LIN {X 0,Y 330.003,Z 389.602,A -85,B 0,C 180,E1 16570.474,E2 16570.474} C_VEL
LIN {X 0,Y 329.994,Z 389.602,A -85,B 0,C 180,E1 16566.088,E2 16566.088} C_VEL
LIN {X 0,Y 329.994,Z 389.603,A -85,B 0,C 180,E1 16561.737,E2 16561.737} C_VEL
LIN {X 0,Y 329.99,Z 389.605,A -85,B 0,C 180,E1 16557.569,E2 16557.569} C_VEL
LIN {X 0,Y 329.99,Z 389.606,A -85,B 0,C 180,E1 16553.389,E2 16553.389} C_VEL
LIN {X 0,Y 330.035,Z 389.884,A -85,B 0,C 180,E1 16551.112,E2 16551.112} C_VEL
LIN {X 0,Y 331.913,Z 393.87,A -85,B 0,C 180,E1 16548.356,E2 16548.356} C_VEL
LIN {X 0,Y 333.849,Z 395.924,A -85,B 0,C 180,E1 16546.667,E2 16546.667} C_VEL
LIN {X 0,Y 335.511,Z 399.399,A -85,B 0,C 180,E1 16544.899,E2 16544.899} C_VEL
LIN {X 0,Y 337.269,Z 401.236,A -85,B 0,C 180,E1 16543.643,E2 16543.643} C_VEL
LIN {X 0,Y 339.377,Z 405.391,A -85,B 0,C 180,E1 16541.803,E2 16541.803} C_VEL
LIN {X 0,Y 340.634,Z 406.903,A -85,B 0,C 180,E1 16540.985,E2 16540.985} C_VEL
LIN {X 0,Y 342.868,Z 410.966,A -85,B 0,C 180,E1 16539.338,E2 16539.338} C_VEL
LIN {X 0,Y 343.879,Z 412.519,A -85,B 0,C 180,E1 16538.688,E2 16538.688} C_VEL
LIN {X 0,Y 346.89,Z 417.767,A -85,B 0,C 180,E1 16536.742,E2 16536.742} C_VEL
LIN {X 0,Y 349.987,Z 423.502,A -85,B 0,C 180,E1 16534.807,E2 16534.807} C_VEL
LIN {X 0,Y 354.378,Z 431.199,A -85,B 0,C 180,E1 16532.438,E2 16532.438} C_VEL
LIN {X 0,Y 356.693,Z 435.152,A -85,B 0,C 180,E1 16531.404,E2 16531.404} C_VEL
LIN {X 0,Y 367.796,Z 451.469,A -85,B 0,C 180,E1 16528.171,E2 16528.171} C_VEL
LIN {X 0,Y 378.595,Z 468.691,A -85,B 0,C 180,E1 16525.38,E2 16525.38} C_VEL
LIN {X 0,Y 387.714,Z 484.728,A -85,B 0,C 180,E1 16523.218,E2 16523.218} C_VEL
LIN {X 0,Y 388.835,Z 502.462,A -85,B 0,C 180,E1 16522.506,E2 16522.506} C_VEL
LIN {X 0,Y 377.647,Z 727.437,A -85,B 0,C 180,E1 16517.928,E2 16517.928} C_VEL
LIN {X 0,Y 375.867,Z 750.219,A -85,B 0,C 180,E1 16517.346,E2 16517.346} C_VEL
LIN {X 0,Y 373.011,Z 772.099,A -85,B 0,C 180,E1 16516.574,E2 16516.574} C_VEL
LIN {X 0,Y 369.512,Z 793.175,A -85,B 0,C 180,E1 16515.585,E2 16515.585} C_VEL
LIN {X 0,Y 365.582,Z 813.65,A -85,B 0,C 180,E1 16514.349,E2 16514.349} C_VEL
LIN {X 0,Y 361.114,Z 833.926,A -85,B 0,C 180,E1 16512.8,E2 16512.8} C_VEL
LIN {X 0,Y 356.36,Z 853.921,A -85,B 0,C 180,E1 16510.926,E2 16510.926} C_VEL
LIN {X 0,Y 351.681,Z 872.496,A -85,B 0,C 180,E1 16508.831,E2 16508.831} C_VEL
LIN {X 0,Y 347.018,Z 890.477,A -85,B 0,C 180,E1 16506.405,E2 16506.405} C_VEL
LIN {X 0,Y 342.617,Z 907.379,A -85,B 0,C 180,E1 16503.672,E2 16503.672} C_VEL
LIN {X 0,Y 338.702,Z 922.893,A -85,B 0,C 180,E1 16500.708,E2 16500.708} C_VEL
LIN {X 0,Y 335.376,Z 937.045,A -85,B 0,C 180,E1 16497.52,E2 16497.52} C_VEL
LIN {X 0,Y 332.739,Z 949.762,A -85,B 0,C 180,E1 16494.119,E2 16494.119} C_VEL
LIN {X 0,Y 330.896,Z 960.4,A -85,B 0,C 180,E1 16490.702,E2 16490.702} C_VEL
LIN {X 0,Y 329.651,Z 970.124,A -85,B 0,C 180,E1 16486.927,E2 16486.927} C_VEL
LIN {X 0,Y 329.068,Z 977.534,A -85,B 0,C 180,E1 16483.351,E2 16483.351} C_VEL
LIN {X 0,Y 328.923,Z 982.817,A -85,B 0,C 180,E1 16479.974,E2 16479.974} C_VEL
LIN {X 0,Y 329.013,Z 986.82,A -85,B 0,C 180,E1 16476.456,E2 16476.456} C_VEL
LIN {X 0,Y 329.151,Z 988.897,A -85,B 0,C 180,E1 16473.309,E2 16473.309} C_VEL
LIN {X 0,Y 329.21,Z 989.725,A -85,B 0,C 180,E1 16470.001,E2 16470.001} C_VEL
LIN {X 0,Y 329.151,Z 988.895,A -85,B 0,C 180,E1 16466.692,E2 16466.692} C_VEL
LIN {X 0,Y 328.997,Z 986.675,A -85,B 0,C 180,E1 16463.37,E2 16463.37} C_VEL
LIN {X 0,Y 328.923,Z 982.807,A -85,B 0,C 180,E1 16460.024,E2 16460.024} C_VEL
LIN {X 0,Y 329.07,Z 977.532,A -85,B 0,C 180,E1 16456.651,E2 16456.651} C_VEL
LIN {X 0,Y 329.651,Z 970.118,A -85,B 0,C 180,E1 16453.074,E2 16453.074} C_VEL
LIN {X 0,Y 330.896,Z 960.39,A -85,B 0,C 180,E1 16449.299,E2 16449.299} C_VEL
LIN {X 0,Y 332.738,Z 949.749,A -85,B 0,C 180,E1 16445.882,E2 16445.882} C_VEL
LIN {X 0,Y 335.375,Z 937.03,A -85,B 0,C 180,E1 16442.481,E2 16442.481} C_VEL
LIN {X 0,Y 338.698,Z 922.869,A -85,B 0,C 180,E1 16439.293,E2 16439.293} C_VEL
LIN {X 0,Y 342.871,Z 906.346,A -85,B 0,C 180,E1 16436.157,E2 16436.157} C_VEL
LIN {X 0,Y 347.175,Z 889.779,A -85,B 0,C 180,E1 16433.502,E2 16433.502} C_VEL
LIN {X 0,Y 351.824,Z 871.877,A -85,B 0,C 180,E1 16431.098,E2 16431.098} C_VEL
LIN {X 0,Y 356.539,Z 853.078,A -85,B 0,C 180,E1 16428.994,E2 16428.994} C_VEL
LIN {X 0,Y 361.35,Z 832.734,A -85,B 0,C 180,E1 16427.109,E2 16427.109} C_VEL
LIN {X 0,Y 365.746,Z 812.621,A -85,B 0,C 180,E1 16425.592,E2 16425.592} C_VEL
LIN {X 0,Y 369.498,Z 793.027,A -85,B 0,C 180,E1 16424.414,E2 16424.414} C_VEL
LIN {X 0,Y 373.124,Z 771.026,A -85,B 0,C 180,E1 16423.389,E2 16423.389} C_VEL
LIN {X 0,Y 375.954,Z 748.774,A -85,B 0,C 180,E1 16422.62,E2 16422.62} C_VEL
LIN {X 0,Y 377.683,Z 725.948,A -85,B 0,C 180,E1 16422.047,E2 16422.047} C_VEL
LIN {X 0,Y 388.788,Z 501.937,A -85,B 0,C 180,E1 16417.493,E2 16417.493} C_VEL
LIN {X 0,Y 387.449,Z 484.37,A -85,B 0,C 180,E1 16416.754,E2 16416.754} C_VEL
LIN {X 0,Y 378.029,Z 467.853,A -85,B 0,C 180,E1 16414.518,E2 16414.518} C_VEL
LIN {X 0,Y 367.562,Z 451.191,A -85,B 0,C 180,E1 16411.806,E2 16411.806} C_VEL
LIN {X 0,Y 357.829,Z 436.979,A -85,B 0,C 180,E1 16408.999,E2 16408.999} C_VEL
LIN {X 0,Y 355.149,Z 432.88,A -85,B 0,C 180,E1 16408.044,E2 16408.044} C_VEL
LIN {X 0,Y 350.821,Z 424.899,A -85,B 0,C 180,E1 16405.671,E2 16405.671} C_VEL
LIN {X 0,Y 348.088,Z 420.021,A -85,B 0,C 180,E1 16404.072,E2 16404.072} C_VEL
LIN {X 0,Y 345.773,Z 415.852,A -85,B 0,C 180,E1 16402.618,E2 16402.618} C_VEL
LIN {X 0,Y 343.042,Z 411.157,A -85,B 0,C 180,E1 16400.829,E2 16400.829} C_VEL
LIN {X 0,Y 340.721,Z 407.214,A -85,B 0,C 180,E1 16399.187,E2 16399.187} C_VEL
LIN {X 0,Y 339.77,Z 405.832,A -85,B 0,C 180,E1 16398.531,E2 16398.531} C_VEL
LIN {X 0,Y 337.632,Z 402.353,A -85,B 0,C 180,E1 16396.87,E2 16396.87} C_VEL
LIN {X 0,Y 336.914,Z 400.853,A -85,B 0,C 180,E1 16396.198,E2 16396.198} C_VEL
LIN {X 0,Y 334.245,Z 397.275,A -85,B 0,C 180,E1 16394.022,E2 16394.022} C_VEL
LIN {X 0,Y 333.382,Z 395.238,A -85,B 0,C 180,E1 16392.999,E2 16392.999} C_VEL
LIN {X 0,Y 330.581,Z 391.815,A -85,B 0,C 180,E1 16390.279,E2 16390.279} C_VEL
LIN {X 0,Y 330.047,Z 389.915,A -85,B 0,C 180,E1 16389.063,E2 16389.063} C_VEL
LIN {X 0,Y 330.015,Z 389.619,A -85,B 0,C 180,E1 16385.389,E2 16385.389} C_VEL
LIN {X 0,Y 330.027,Z 389.618,A -85,B 0,C 180,E1 16381.041,E2 16381.041} C_VEL
LIN {X 0,Y 330.014,Z 389.616,A -85,B 0,C 180,E1 16376.7,E2 16376.7} C_VEL
LIN {X 0,Y 330.005,Z 389.613,A -85,B 0,C 180,E1 16372.339,E2 16372.339} C_VEL
LIN {X 0,Y 330.004,Z 389.612,A -85,B 0,C 180,E1 16368.105,E2 16368.105} C_VEL
LIN {X 0,Y 330.002,Z 389.614,A -85,B 0,C 180,E1 16363.813,E2 16363.813} C_VEL
LIN {X 0,Y 330.043,Z 389.821,A -85,B 0,C 180,E1 16361.085,E2 16361.085} C_VEL
LIN {X 0,Y 332.016,Z 393.974,A -85,B 0,C 180,E1 16358.073,E2 16358.073} C_VEL
LIN {X 0,Y 333.668,Z 395.964,A -85,B 0,C 180,E1 16356.512,E2 16356.512} C_VEL
LIN {X 0,Y 335.446,Z 399.475,A -85,B 0,C 180,E1 16354.582,E2 16354.582} C_VEL
LIN {X 0,Y 336.766,Z 401.01,A -85,B 0,C 180,E1 16353.554,E2 16353.554} C_VEL
LIN {X 0,Y 338.824,Z 405.069,A -85,B 0,C 180,E1 16351.633,E2 16351.633} C_VEL
LIN {X 0,Y 339.913,Z 406.594,A -85,B 0,C 180,E1 16350.872,E2 16350.872} C_VEL
LIN {X 0,Y 343.38,Z 410.881,A -85,B 0,C 180,E1 16349.461,E2 16349.461} C_VEL
LIN {X 0,Y 345.144,Z 412.815,A -85,B 0,C 180,E1 16348.813,E2 16348.813} C_VEL
LIN {X 0,Y 350.069,Z 418.726,A -85,B 0,C 180,E1 16347.085,E2 16347.085} C_VEL
LIN {X 0,Y 355.033,Z 424.875,A -85,B 0,C 180,E1 16345.474,E2 16345.474} C_VEL
LIN {X 0,Y 359.624,Z 430.701,A -85,B 0,C 180,E1 16344.081,E2 16344.081} C_VEL
LIN {X 0,Y 366.377,Z 439.666,A -85,B 0,C 180,E1 16342.167,E2 16342.167} C_VEL
LIN {X 0,Y 375.291,Z 452.29,A -85,B 0,C 180,E1 16339.853,E2 16339.853} C_VEL
LIN {X 0,Y 385.053,Z 467.432,A -85,B 0,C 180,E1 16337.535,E2 16337.535} C_VEL
LIN {X 0,Y 387.229,Z 471.318,A -85,B 0,C 180,E1 16337.036,E2 16337.036} C_VEL
LIN {X 0,Y 378.765,Z 667.93,A -85,B 0,C 180,E1 16333.284,E2 16333.284} C_VEL
LIN {X 0,Y 377.338,Z 688.38,A -85,B 0,C 180,E1 16332.637,E2 16332.637} C_VEL
LIN {X 0,Y 375.079,Z 708.985,A -85,B 0,C 180,E1 16331.72,E2 16331.72} C_VEL
LIN {X 0,Y 372.311,Z 727.719,A -85,B 0,C 180,E1 16330.63,E2 16330.63} C_VEL
LIN {X 0,Y 368.842,Z 746.294,A -85,B 0,C 180,E1 16329.264,E2 16329.264} C_VEL
LIN {X 0,Y 364.892,Z 763.906,A -85,B 0,C 180,E1 16327.661,E2 16327.661} C_VEL
LIN {X 0,Y 360.603,Z 780.679,A -85,B 0,C 180,E1 16325.801,E2 16325.801} C_VEL
LIN {X 0,Y 356.094,Z 796.544,A -85,B 0,C 180,E1 16323.675,E2 16323.675} C_VEL
LIN {X 0,Y 351.629,Z 810.958,A -85,B 0,C 180,E1 16321.352,E2 16321.352} C_VEL
LIN {X 0,Y 347.209,Z 824.285,A -85,B 0,C 180,E1 16318.741,E2 16318.741} C_VEL
LIN {X 0,Y 343.088,Z 836.219,A -85,B 0,C 180,E1 16315.918,E2 16315.918} C_VEL
LIN {X 0,Y 339.249,Z 847.309,A -85,B 0,C 180,E1 16312.705,E2 16312.705} C_VEL
LIN {X 0,Y 336.142,Z 856.384,A -85,B 0,C 180,E1 16309.451,E2 16309.451} C_VEL
LIN {X 0,Y 333.701,Z 864.021,A -85,B 0,C 180,E1 16305.999,E2 16305.999} C_VEL
LIN {X 0,Y 331.861,Z 870.159,A -85,B 0,C 180,E1 16302.35,E2 16302.35} C_VEL
LIN {X 0,Y 330.727,Z 874.547,A -85,B 0,C 180,E1 16298.661,E2 16298.661} C_VEL
LIN {X 0,Y 330.097,Z 877.302,A -85,B 0,C 180,E1 16295.038,E2 16295.038} C_VEL
LIN {X 0,Y 329.836,Z 878.634,A -85,B 0,C 180,E1 16291.215,E2 16291.215} C_VEL
LIN {X 0,Y 329.887,Z 878.441,A -85,B 0,C 180,E1 16287.568,E2 16287.568} C_VEL
LIN {X 0,Y 330.224,Z 876.777,A -85,B 0,C 180,E1 16283.917,E2 16283.917} C_VEL
LIN {X 0,Y 330.978,Z 873.537,A -85,B 0,C 180,E1 16280.261,E2 16280.261} C_VEL
LIN {X 0,Y 331.265,Z 872.383,A -85,B 0,C 180,E1 16279.251,E2 16279.251} C_VEL
LIN {X 0,Y 330.73,Z 870.915,A -85,B 0,C 180,E1 16277.935,E2 16277.935} C_VEL
LIN {X 0,Y 326.334,Z 866.853,A -85,B 0,C 180,E1 16274.375,E2 16274.375} C_VEL
LIN {X 0,Y 326.261,Z 864.89,A -85,B 0,C 180,E1 16273.256,E2 16273.256} C_VEL
LIN {X 0,Y 329.077,Z 856.714,A -85,B 0,C 180,E1 16269.55,E2 16269.55} C_VEL
LIN {X 0,Y 332.446,Z 847.383,A -85,B 0,C 180,E1 16266.235,E2 16266.235} C_VEL
LIN {X 0,Y 336.356,Z 836.657,A -85,B 0,C 180,E1 16263.141,E2 16263.141} C_VEL
LIN {X 0,Y 341,Z 823.745,A -85,B 0,C 180,E1 16260.104,E2 16260.104} C_VEL
LIN {X 0,Y 345.699,Z 810.039,A -85,B 0,C 180,E1 16257.458,E2 16257.458} C_VEL
LIN {X 0,Y 350.459,Z 795.347,A -85,B 0,C 180,E1 16255.112,E2 16255.112} C_VEL
LIN {X 0,Y 355.212,Z 779.012,A -85,B 0,C 180,E1 16252.964,E2 16252.964} C_VEL
LIN {X 0,Y 359.544,Z 762.288,A -85,B 0,C 180,E1 16251.158,E2 16251.158} C_VEL
LIN {X 0,Y 363.644,Z 744.081,A -85,B 0,C 180,E1 16249.546,E2 16249.546} C_VEL
LIN {X 0,Y 367.152,Z 725.385,A -85,B 0,C 180,E1 16248.21,E2 16248.21} C_VEL
LIN {X 0,Y 370.075,Z 705.564,A -85,B 0,C 180,E1 16247.095,E2 16247.095} C_VEL
LIN {X 0,Y 372.251,Z 684.715,A -85,B 0,C 180,E1 16246.225,E2 16246.225} C_VEL
LIN {X 0,Y 373.521,Z 664.33,A -85,B 0,C 180,E1 16245.638,E2 16245.638} C_VEL
LIN {X 0,Y 381.975,Z 474.612,A -85,B 0,C 180,E1 16241.984,E2 16241.984} C_VEL
LIN {X 0,Y 372.325,Z 459.299,A -85,B 0,C 180,E1 16239.628,E2 16239.628} C_VEL
LIN {X 0,Y 363.175,Z 446.134,A -85,B 0,C 180,E1 16237.179,E2 16237.179} C_VEL
LIN {X 0,Y 354.803,Z 434.794,A -85,B 0,C 180,E1 16234.698,E2 16234.698} C_VEL
LIN {X 0,Y 349.127,Z 427.883,A -85,B 0,C 180,E1 16232.868,E2 16232.868} C_VEL
LIN {X 0,Y 345.683,Z 423.571,A -85,B 0,C 180,E1 16231.667,E2 16231.667} C_VEL
LIN {X 0,Y 341.36,Z 418.367,A -85,B 0,C 180,E1 16230.058,E2 16230.058} C_VEL
LIN {X 0,Y 337.475,Z 413.639,A -85,B 0,C 180,E1 16228.49,E2 16228.49} C_VEL
LIN {X 0,Y 332.939,Z 408.828,A -85,B 0,C 180,E1 16226.51,E2 16226.51} C_VEL
LIN {X 0,Y 331.894,Z 406.975,A -85,B 0,C 180,E1 16225.71,E2 16225.71} C_VEL
LIN {X 0,Y 329.62,Z 403.66,A -85,B 0,C 180,E1 16223.604,E2 16223.604} C_VEL
LIN {X 0,Y 328.802,Z 401.717,A -85,B 0,C 180,E1 16222.53,E2 16222.53} C_VEL
LIN {X 0,Y 326.275,Z 398.234,A -85,B 0,C 180,E1 16219.7,E2 16219.7} C_VEL
LIN {X 0,Y 325.448,Z 396.214,A -85,B 0,C 180,E1 16218.263,E2 16218.263} C_VEL
LIN {X 0,Y 322.129,Z 390.882,A -85,B 0,C 180,E1 16211.458,E2 16211.458} C_VEL
LIN {X 0,Y 322.106,Z 390.591,A -85,B 0,C 180,E1 16207.133,E2 16207.133} C_VEL
LIN {X 0,Y 322.074,Z 390.595,A -85,B 0,C 180,E1 16202.669,E2 16202.669} C_VEL
LIN {X 0,Y 322.11,Z 390.849,A -85,B 0,C 180,E1 16198.577,E2 16198.577} C_VEL
LIN {X 0,Y 322.685,Z 392.882,A -85,B 0,C 180,E1 16195.914,E2 16195.914} C_VEL
LIN {X 0,Y 326.065,Z 397.027,A -85,B 0,C 180,E1 16191.003,E2 16191.003} C_VEL
LIN {X 0,Y 327.843,Z 400.664,A -85,B 0,C 180,E1 16188.567,E2 16188.567} C_VEL
LIN {X 0,Y 329.725,Z 402.803,A -85,B 0,C 180,E1 16186.855,E2 16186.855} C_VEL
LIN {X 0,Y 331.523,Z 406.341,A -85,B 0,C 180,E1 16184.968,E2 16184.968} C_VEL
LIN {X 0,Y 333.073,Z 408.159,A -85,B 0,C 180,E1 16183.789,E2 16183.789} C_VEL
LIN {X 0,Y 335.23,Z 412.194,A -85,B 0,C 180,E1 16181.93,E2 16181.93} C_VEL
LIN {X 0,Y 336.394,Z 413.89,A -85,B 0,C 180,E1 16181.097,E2 16181.097} C_VEL
LIN {X 0,Y 338.669,Z 417.763,A -85,B 0,C 180,E1 16179.432,E2 16179.432} C_VEL
LIN {X 0,Y 342.389,Z 424.435,A -85,B 0,C 180,E1 16176.896,E2 16176.896} C_VEL
LIN {X 0,Y 347.188,Z 432.781,A -85,B 0,C 180,E1 16174.132,E2 16174.132} C_VEL
LIN {X 0,Y 356.696,Z 446.221,A -85,B 0,C 180,E1 16170.985,E2 16170.985} C_VEL
LIN {X 0,Y 365.616,Z 459.773,A -85,B 0,C 180,E1 16168.374,E2 16168.374} C_VEL
LIN {X 0,Y 375.477,Z 475.857,A -85,B 0,C 180,E1 16165.769,E2 16165.769} C_VEL
LIN {X 0,Y 382.746,Z 489.077,A -85,B 0,C 180,E1 16163.978,E2 16163.978} C_VEL
LIN {X 0,Y 383.574,Z 503.771,A -85,B 0,C 180,E1 16163.386,E2 16163.386} C_VEL
LIN {X 0,Y 371.975,Z 727.631,A -85,B 0,C 180,E1 16158.791,E2 16158.791} C_VEL
LIN {X 0,Y 370.089,Z 750.508,A -85,B 0,C 180,E1 16158.196,E2 16158.196} C_VEL
LIN {X 0,Y 366.998,Z 772.907,A -85,B 0,C 180,E1 16157.383,E2 16157.383} C_VEL
LIN {X 0,Y 363.301,Z 793.934,A -85,B 0,C 180,E1 16156.365,E2 16156.365} C_VEL
LIN {X 0,Y 359.188,Z 814.241,A -85,B 0,C 180,E1 16155.103,E2 16155.103} C_VEL
LIN {X 0,Y 354.664,Z 833.933,A -85,B 0,C 180,E1 16153.571,E2 16153.571} C_VEL
LIN {X 0,Y 349.878,Z 853.081,A -85,B 0,C 180,E1 16151.743,E2 16151.743} C_VEL
LIN {X 0,Y 344.762,Z 872.403,A -85,B 0,C 180,E1 16149.518,E2 16149.518} C_VEL
LIN {X 0,Y 339.95,Z 890.082,A -85,B 0,C 180,E1 16147.077,E2 16147.077} C_VEL
LIN {X 0,Y 335.348,Z 906.863,A -85,B 0,C 180,E1 16144.296,E2 16144.296} C_VEL
LIN {X 0,Y 331.23,Z 922.242,A -85,B 0,C 180,E1 16141.276,E2 16141.276} C_VEL
LIN {X 0,Y 327.741,Z 936.279,A -85,B 0,C 180,E1 16138.02,E2 16138.02} C_VEL
LIN {X 0,Y 324.964,Z 948.937,A -85,B 0,C 180,E1 16134.541,E2 16134.541} C_VEL
LIN {X 0,Y 322.944,Z 960.005,A -85,B 0,C 180,E1 16130.856,E2 16130.856} C_VEL
LIN {X 0,Y 321.716,Z 969.122,A -85,B 0,C 180,E1 16127.171,E2 16127.171} C_VEL
LIN {X 0,Y 321.122,Z 976.457,A -85,B 0,C 180,E1 16123.504,E2 16123.504} C_VEL
LIN {X 0,Y 320.989,Z 981.691,A -85,B 0,C 180,E1 16120.045,E2 16120.045} C_VEL
LIN {X 0,Y 321.103,Z 985.614,A -85,B 0,C 180,E1 16116.436,E2 16116.436} C_VEL
LIN {X 0,Y 321.257,Z 987.645,A -85,B 0,C 180,E1 16113.212,E2 16113.212} C_VEL
LIN {X 0,Y 321.313,Z 988.379,A -85,B 0,C 180,E1 16109.822,E2 16109.822} C_VEL
LIN {X 0,Y 321.252,Z 987.562,A -85,B 0,C 180,E1 16106.611,E2 16106.611} C_VEL
LIN {X 0,Y 321.068,Z 985.328,A -85,B 0,C 180,E1 16103.205,E2 16103.205} C_VEL
LIN {X 0,Y 320.994,Z 981.444,A -85,B 0,C 180,E1 16099.775,E2 16099.775} C_VEL
LIN {X 0,Y 321.142,Z 976.046,A -85,B 0,C 180,E1 16096.261,E2 16096.261} C_VEL
LIN {X 0,Y 321.756,Z 968.707,A -85,B 0,C 180,E1 16092.646,E2 16092.646} C_VEL
LIN {X 0,Y 323.109,Z 958.955,A -85,B 0,C 180,E1 16088.776,E2 16088.776} C_VEL
LIN {X 0,Y 325.09,Z 948.289,A -85,B 0,C 180,E1 16085.277,E2 16085.277} C_VEL
LIN {X 0,Y 327.927,Z 935.494,A -85,B 0,C 180,E1 16081.783,E2 16081.783} C_VEL
LIN {X 0,Y 331.439,Z 921.369,A -85,B 0,C 180,E1 16078.545,E2 16078.545} C_VEL
LIN {X 0,Y 335.871,Z 904.821,A -85,B 0,C 180,E1 16075.353,E2 16075.353} C_VEL
LIN {X 0,Y 340.419,Z 888.284,A -85,B 0,C 180,E1 16072.667,E2 16072.667} C_VEL
LIN {X 0,Y 345.318,Z 870.306,A -85,B 0,C 180,E1 16070.221,E2 16070.221} C_VEL
LIN {X 0,Y 350.265,Z 851.458,A -85,B 0,C 180,E1 16068.095,E2 16068.095} C_VEL
LIN {X 0,Y 355.308,Z 831.044,A -85,B 0,C 180,E1 16066.197,E2 16066.197} C_VEL
LIN {X 0,Y 359.883,Z 810.815,A -85,B 0,C 180,E1 16064.671,E2 16064.671} C_VEL
LIN {X 0,Y 363.792,Z 791.147,A -85,B 0,C 180,E1 16063.489,E2 16063.489} C_VEL
LIN {X 0,Y 367.482,Z 769.334,A -85,B 0,C 180,E1 16062.48,E2 16062.48} C_VEL
LIN {X 0,Y 370.426,Z 746.466,A -85,B 0,C 180,E1 16061.697,E2 16061.697} C_VEL
LIN {X 0,Y 372.158,Z 723.573,A -85,B 0,C 180,E1 16061.128,E2 16061.128} C_VEL
LIN {X 0,Y 383.568,Z 502.348,A -85,B 0,C 180,E1 16056.595,E2 16056.595} C_VEL
LIN {X 0,Y 382.472,Z 488.457,A -85,B 0,C 180,E1 16055.982,E2 16055.982} C_VEL
LIN {X 0,Y 373.484,Z 472.672,A -85,B 0,C 180,E1 16053.768,E2 16053.768} C_VEL
LIN {X 0,Y 364.034,Z 457.35,A -85,B 0,C 180,E1 16051.226,E2 16051.226} C_VEL
LIN {X 0,Y 353.368,Z 441.428,A -85,B 0,C 180,E1 16048.014,E2 16048.014} C_VEL
LIN {X 0,Y 346.589,Z 431.867,A -85,B 0,C 180,E1 16045.64,E2 16045.64} C_VEL
LIN {X 0,Y 341.564,Z 422.688,A -85,B 0,C 180,E1 16042.549,E2 16042.549} C_VEL
LIN {X 0,Y 338.315,Z 417.33,A -85,B 0,C 180,E1 16040.41,E2 16040.41} C_VEL
LIN {X 0,Y 335.627,Z 412.638,A -85,B 0,C 180,E1 16038.408,E2 16038.408} C_VEL
LIN {X 0,Y 333.288,Z 408.82,A -85,B 0,C 180,E1 16036.558,E2 16036.558} C_VEL
LIN {X 0,Y 332.533,Z 407.434,A -85,B 0,C 180,E1 16035.879,E2 16035.879} C_VEL
LIN {X 0,Y 329.983,Z 403.734,A -85,B 0,C 180,E1 16033.67,E2 16033.67} C_VEL
LIN {X 0,Y 329.27,Z 402.069,A -85,B 0,C 180,E1 16032.807,E2 16032.807} C_VEL
LIN {X 0,Y 326.424,Z 398.309,A -85,B 0,C 180,E1 16029.876,E2 16029.876} C_VEL
LIN {X 0,Y 325.681,Z 396.429,A -85,B 0,C 180,E1 16028.652,E2 16028.652} C_VEL
LIN {X 0,Y 322.307,Z 391.747,A -85,B 0,C 180,E1 16023.201,E2 16023.201} C_VEL
LIN {X 0,Y 322.095,Z 390.658,A -85,B 0,C 180,E1 16021.067,E2 16021.067} C_VEL
LIN {X 0,Y 322.07,Z 390.606,A -85,B 0,C 180,E1 16016.618,E2 16016.618} C_VEL
LIN {X 0,Y 322.066,Z 390.602,A -85,B 0,C 180,E1 16012.328,E2 16012.328} C_VEL
LIN {X 0,Y 322.102,Z 390.844,A -85,B 0,C 180,E1 16008.177,E2 16008.177} C_VEL
LIN {X 0,Y 323.492,Z 394.247,A -85,B 0,C 180,E1 16004.033,E2 16004.033} C_VEL
LIN {X 0,Y 325.894,Z 396.96,A -85,B 0,C 180,E1 16000.835,E2 16000.835} C_VEL
LIN {X 0,Y 327.646,Z 400.558,A -85,B 0,C 180,E1 15998.33,E2 15998.33} C_VEL
LIN {X 0,Y 329.264,Z 402.536,A -85,B 0,C 180,E1 15996.748,E2 15996.748} C_VEL
LIN {X 0,Y 331.005,Z 406.037,A -85,B 0,C 180,E1 15994.791,E2 15994.791} C_VEL
LIN {X 0,Y 332.379,Z 407.811,A -85,B 0,C 180,E1 15993.681,E2 15993.681} C_VEL
LIN {X 0,Y 335.997,Z 412.323,A -85,B 0,C 180,E1 15991.954,E2 15991.954} C_VEL
LIN {X 0,Y 337.813,Z 414.198,A -85,B 0,C 180,E1 15991.203,E2 15991.203} C_VEL
LIN {X 0,Y 341.657,Z 418.632,A -85,B 0,C 180,E1 15989.68,E2 15989.68} C_VEL
LIN {X 0,Y 347.621,Z 425.939,A -85,B 0,C 180,E1 15987.51,E2 15987.51} C_VEL
LIN {X 0,Y 352.74,Z 432.388,A -85,B 0,C 180,E1 15985.809,E2 15985.809} C_VEL
LIN {X 0,Y 359.408,Z 440.965,A -85,B 0,C 180,E1 15983.773,E2 15983.773} C_VEL
LIN {X 0,Y 369.804,Z 455.557,A -85,B 0,C 180,E1 15980.901,E2 15980.901} C_VEL
LIN {X 0,Y 380.14,Z 471.616,A -85,B 0,C 180,E1 15978.333,E2 15978.333} C_VEL
LIN {X 0,Y 381.977,Z 475.055,A -85,B 0,C 180,E1 15977.89,E2 15977.89} C_VEL
LIN {X 0,Y 373.244,Z 668.782,A -85,B 0,C 180,E1 15974.157,E2 15974.157} C_VEL
LIN {X 0,Y 371.754,Z 689.342,A -85,B 0,C 180,E1 15973.501,E2 15973.501} C_VEL
LIN {X 0,Y 369.411,Z 709.933,A -85,B 0,C 180,E1 15972.577,E2 15972.577} C_VEL
LIN {X 0,Y 366.612,Z 728.319,A -85,B 0,C 180,E1 15971.503,E2 15971.503} C_VEL
LIN {X 0,Y 363.002,Z 746.957,A -85,B 0,C 180,E1 15970.125,E2 15970.125} C_VEL
LIN {X 0,Y 358.879,Z 764.745,A -85,B 0,C 180,E1 15968.497,E2 15968.497} C_VEL
LIN {X 0,Y 354.253,Z 782.156,A -85,B 0,C 180,E1 15966.546,E2 15966.546} C_VEL
LIN {X 0,Y 349.563,Z 797.978,A -85,B 0,C 180,E1 15964.391,E2 15964.391} C_VEL
LIN {X 0,Y 344.909,Z 812.369,A -85,B 0,C 180,E1 15962.035,E2 15962.035} C_VEL
LIN {X 0,Y 340.03,Z 826.469,A -85,B 0,C 180,E1 15959.213,E2 15959.213} C_VEL
LIN {X 0,Y 335.686,Z 838.42,A -85,B 0,C 180,E1 15956.292,E2 15956.292} C_VEL
LIN {X 0,Y 331.946,Z 848.664,A -85,B 0,C 180,E1 15953.237,E2 15953.237} C_VEL
LIN {X 0,Y 328.672,Z 857.724,A -85,B 0,C 180,E1 15949.918,E2 15949.918} C_VEL
LIN {X 0,Y 326.079,Z 865.367,A -85,B 0,C 180,E1 15946.383,E2 15946.383} C_VEL
LIN {X 0,Y 324.121,Z 871.502,A -85,B 0,C 180,E1 15942.65,E2 15942.65} C_VEL
LIN {X 0,Y 322.913,Z 875.851,A -85,B 0,C 180,E1 15938.905,E2 15938.905} C_VEL
LIN {X 0,Y 322.219,Z 878.681,A -85,B 0,C 180,E1 15935.074,E2 15935.074} C_VEL
LIN {X 0,Y 321.947,Z 879.962,A -85,B 0,C 180,E1 15931.245,E2 15931.245} C_VEL
LIN {X 0,Y 322.002,Z 879.769,A -85,B 0,C 180,E1 15927.508,E2 15927.508} C_VEL
LIN {X 0,Y 322.366,Z 878.107,A -85,B 0,C 180,E1 15923.768,E2 15923.768} C_VEL
LIN {X 0,Y 323.175,Z 874.873,A -85,B 0,C 180,E1 15920.023,E2 15920.023} C_VEL
LIN {X 0,Y 324.55,Z 870.04,A -85,B 0,C 180,E1 15916.278,E2 15916.278} C_VEL
LIN {X 0,Y 326.261,Z 864.89,A -85,B 0,C 180,E1 15913.256,E2 15913.256} C_VEL
LIN {X 0,Y 326.136,Z 862.521,A -85,B 0,C 180,E1 15911.962,E2 15911.962} C_VEL
LIN {X 0,Y 323.027,Z 856.609,A -85,B 0,C 180,E1 15908.609,E2 15908.609} C_VEL
LIN {X 0,Y 323.355,Z 853.579,A -85,B 0,C 180,E1 15907.336,E2 15907.336} C_VEL
LIN {X 0,Y 327.153,Z 843.633,A -85,B 0,C 180,E1 15904.087,E2 15904.087} C_VEL
LIN {X 0,Y 331.661,Z 831.852,A -85,B 0,C 180,E1 15900.959,E2 15900.959} C_VEL
LIN {X 0,Y 336.545,Z 818.584,A -85,B 0,C 180,E1 15898.077,E2 15898.077} C_VEL
LIN {X 0,Y 341.415,Z 804.691,A -85,B 0,C 180,E1 15895.586,E2 15895.586} C_VEL
LIN {X 0,Y 346.541,Z 788.705,A -85,B 0,C 180,E1 15893.228,E2 15893.228} C_VEL
LIN {X 0,Y 351.276,Z 772.183,A -85,B 0,C 180,E1 15891.234,E2 15891.234} C_VEL
LIN {X 0,Y 355.666,Z 754.807,A -85,B 0,C 180,E1 15889.508,E2 15889.508} C_VEL
LIN {X 0,Y 359.575,Z 736.634,A -85,B 0,C 180,E1 15888.034,E2 15888.034} C_VEL
LIN {X 0,Y 362.938,Z 717.632,A -85,B 0,C 180,E1 15886.801,E2 15886.801} C_VEL
LIN {X 0,Y 365.627,Z 697.318,A -85,B 0,C 180,E1 15885.791,E2 15885.791} C_VEL
LIN {X 0,Y 367.414,Z 677.439,A -85,B 0,C 180,E1 15885.068,E2 15885.068} C_VEL
LIN {X 0,Y 368.66,Z 651.848,A -85,B 0,C 180,E1 15884.452,E2 15884.452} C_VEL
LIN {X 0,Y 376.813,Z 478.354,A -85,B 0,C 180,E1 15881.104,E2 15881.104} C_VEL
LIN {X 0,Y 367.016,Z 462.764,A -85,B 0,C 180,E1 15878.599,E2 15878.599} C_VEL
LIN {X 0,Y 357.401,Z 449.022,A -85,B 0,C 180,E1 15875.881,E2 15875.881} C_VEL
LIN {X 0,Y 350.443,Z 439.811,A -85,B 0,C 180,E1 15873.707,E2 15873.707} C_VEL
LIN {X 0,Y 346.358,Z 434.657,A -85,B 0,C 180,E1 15872.329,E2 15872.329} C_VEL
LIN {X 0,Y 342.972,Z 430.403,A -85,B 0,C 180,E1 15871.114,E2 15871.114} C_VEL
LIN {X 0,Y 339.038,Z 425.56,A -85,B 0,C 180,E1 15869.603,E2 15869.603} C_VEL
LIN {X 0,Y 334.469,Z 420.152,A -85,B 0,C 180,E1 15867.701,E2 15867.701} C_VEL
LIN {X 0,Y 330.311,Z 415.312,A -85,B 0,C 180,E1 15865.794,E2 15865.794} C_VEL
LIN {X 0,Y 325.432,Z 410.225,A -85,B 0,C 180,E1 15863.283,E2 15863.283} C_VEL
LIN {X 0,Y 324.639,Z 408.535,A -85,B 0,C 180,E1 15862.452,E2 15862.452} C_VEL
LIN {X 0,Y 322.031,Z 404.808,A -85,B 0,C 180,E1 15859.404,E2 15859.404} C_VEL
LIN {X 0,Y 321.339,Z 403.057,A -85,B 0,C 180,E1 15858.129,E2 15858.129} C_VEL
LIN {X 0,Y 317.876,Z 397.555,A -85,B 0,C 180,E1 15851.062,E2 15851.062} C_VEL
LIN {X 0,Y 316.725,Z 396.547,A -85,B 0,C 180,E1 15845.617,E2 15845.617} C_VEL
LIN {X 0,Y 317.485,Z 397.189,A -85,B 0,C 180,E1 15840.181,E2 15840.181} C_VEL
LIN {X 0,Y 318.321,Z 398.376,A -85,B 0,C 180,E1 15837.66,E2 15837.66} C_VEL
LIN {X 0,Y 322.036,Z 403.804,A -85,B 0,C 180,E1 15831.25,E2 15831.25} C_VEL
LIN {X 0,Y 323.774,Z 407.456,A -85,B 0,C 180,E1 15828.782,E2 15828.782} C_VEL
LIN {X 0,Y 325.482,Z 409.252,A -85,B 0,C 180,E1 15827.222,E2 15827.222} C_VEL
LIN {X 0,Y 327.399,Z 413.128,A -85,B 0,C 180,E1 15825.136,E2 15825.136} C_VEL
LIN {X 0,Y 328.876,Z 415.055,A -85,B 0,C 180,E1 15823.939,E2 15823.939} C_VEL
LIN {X 0,Y 331.249,Z 419.231,A -85,B 0,C 180,E1 15821.887,E2 15821.887} C_VEL
LIN {X 0,Y 335.026,Z 425.812,A -85,B 0,C 180,E1 15819.074,E2 15819.074} C_VEL
LIN {X 0,Y 338.065,Z 431.098,A -85,B 0,C 180,E1 15817.113,E2 15817.113} C_VEL
LIN {X 0,Y 345.255,Z 440.94,A -85,B 0,C 180,E1 15814.345,E2 15814.345} C_VEL
LIN {X 0,Y 352.542,Z 451.312,A -85,B 0,C 180,E1 15811.868,E2 15811.868} C_VEL
LIN {X 0,Y 361.63,Z 465.136,A -85,B 0,C 180,E1 15809.098,E2 15809.098} C_VEL
LIN {X 0,Y 371.611,Z 481.692,A -85,B 0,C 180,E1 15806.364,E2 15806.364} C_VEL
LIN {X 0,Y 377.826,Z 493.253,A -85,B 0,C 180,E1 15804.767,E2 15804.767} C_VEL
LIN {X 0,Y 378.401,Z 505.157,A -85,B 0,C 180,E1 15804.289,E2 15804.289} C_VEL
LIN {X 0,Y 366.419,Z 727.442,A -85,B 0,C 180,E1 15799.69,E2 15799.69} C_VEL
LIN {X 0,Y 364.452,Z 750.113,A -85,B 0,C 180,E1 15799.09,E2 15799.09} C_VEL
LIN {X 0,Y 361.223,Z 772.648,A -85,B 0,C 180,E1 15798.263,E2 15798.263} C_VEL
LIN {X 0,Y 357.418,Z 793.388,A -85,B 0,C 180,E1 15797.245,E2 15797.245} C_VEL
LIN {X 0,Y 353.157,Z 813.561,A -85,B 0,C 180,E1 15795.977,E2 15795.977} C_VEL
LIN {X 0,Y 348.288,Z 833.929,A -85,B 0,C 180,E1 15794.372,E2 15794.372} C_VEL
LIN {X 0,Y 343.267,Z 853.02,A -85,B 0,C 180,E1 15792.509,E2 15792.509} C_VEL
LIN {X 0,Y 337.898,Z 872.307,A -85,B 0,C 180,E1 15790.233,E2 15790.233} C_VEL
LIN {X 0,Y 332.792,Z 890.106,A -85,B 0,C 180,E1 15787.705,E2 15787.705} C_VEL
LIN {X 0,Y 328.104,Z 906.391,A -85,B 0,C 180,E1 15784.941,E2 15784.941} C_VEL
LIN {X 0,Y 323.793,Z 921.595,A -85,B 0,C 180,E1 15781.87,E2 15781.87} C_VEL
LIN {X 0,Y 319.953,Z 936.221,A -85,B 0,C 180,E1 15778.357,E2 15778.357} C_VEL
LIN {X 0,Y 317.079,Z 948.658,A -85,B 0,C 180,E1 15774.794,E2 15774.794} C_VEL
LIN {X 0,Y 314.993,Z 959.612,A -85,B 0,C 180,E1 15771.018,E2 15771.018} C_VEL
LIN {X 0,Y 313.742,Z 968.527,A -85,B 0,C 180,E1 15767.239,E2 15767.239} C_VEL
LIN {X 0,Y 313.149,Z 975.971,A -85,B 0,C 180,E1 15763.29,E2 15763.29} C_VEL
LIN {X 0,Y 313.045,Z 981.052,A -85,B 0,C 180,E1 15759.746,E2 15759.746} C_VEL
LIN {X 0,Y 313.22,Z 984.683,A -85,B 0,C 180,E1 15756.047,E2 15756.047} C_VEL
LIN {X 0,Y 313.364,Z 986.55,A -85,B 0,C 180,E1 15752.744,E2 15752.744} C_VEL
LIN {X 0,Y 313.418,Z 986.975,A -85,B 0,C 180,E1 15749.27,E2 15749.27} C_VEL
LIN {X 0,Y 313.332,Z 986.063,A -85,B 0,C 180,E1 15746.159,E2 15746.159} C_VEL
LIN {X 0,Y 313.124,Z 983.621,A -85,B 0,C 180,E1 15742.663,E2 15742.663} C_VEL
LIN {X 0,Y 313.054,Z 979.591,A -85,B 0,C 180,E1 15739.14,E2 15739.14} C_VEL
LIN {X 0,Y 313.277,Z 973.435,A -85,B 0,C 180,E1 15735.251,E2 15735.251} C_VEL
LIN {X 0,Y 314.048,Z 965.965,A -85,B 0,C 180,E1 15731.578,E2 15731.578} C_VEL
LIN {X 0,Y 315.532,Z 956.482,A -85,B 0,C 180,E1 15727.85,E2 15727.85} C_VEL
LIN {X 0,Y 317.898,Z 944.915,A -85,B 0,C 180,E1 15724.079,E2 15724.079} C_VEL
LIN {X 0,Y 320.876,Z 932.652,A -85,B 0,C 180,E1 15720.715,E2 15720.715} C_VEL
LIN {X 0,Y 324.731,Z 918.191,A -85,B 0,C 180,E1 15717.4,E2 15717.4} C_VEL
LIN {X 0,Y 329.077,Z 902.799,A -85,B 0,C 180,E1 15714.424,E2 15714.424} C_VEL
LIN {X 0,Y 334.026,Z 885.789,A -85,B 0,C 180,E1 15711.651,E2 15711.651} C_VEL
LIN {X 0,Y 339.088,Z 868.093,A -85,B 0,C 180,E1 15709.228,E2 15709.228} C_VEL
LIN {X 0,Y 344.302,Z 849.074,A -85,B 0,C 180,E1 15707.085,E2 15707.085} C_VEL
LIN {X 0,Y 349.362,Z 829.361,A -85,B 0,C 180,E1 15705.254,E2 15705.254} C_VEL
LIN {X 0,Y 354.116,Z 809.016,A -85,B 0,C 180,E1 15703.719,E2 15703.719} C_VEL
LIN {X 0,Y 358.482,Z 787.77,A -85,B 0,C 180,E1 15702.452,E2 15702.452} C_VEL
LIN {X 0,Y 362.232,Z 765.852,A -85,B 0,C 180,E1 15701.471,E2 15701.471} C_VEL
LIN {X 0,Y 365.078,Z 743.358,A -85,B 0,C 180,E1 15700.724,E2 15700.724} C_VEL
LIN {X 0,Y 366.902,Z 717.899,A -85,B 0,C 180,E1 15700.112,E2 15700.112} C_VEL
LIN {X 0,Y 378.4,Z 503.584,A -85,B 0,C 180,E1 15695.688,E2 15695.688} C_VEL
LIN {X 0,Y 377.561,Z 492.575,A -85,B 0,C 180,E1 15695.191,E2 15695.191} C_VEL
LIN {X 0,Y 367.764,Z 475.246,A -85,B 0,C 180,E1 15692.661,E2 15692.661} C_VEL
LIN {X 0,Y 358.406,Z 460.185,A -85,B 0,C 180,E1 15690.003,E2 15690.003} C_VEL
LIN {X 0,Y 349.307,Z 446.653,A -85,B 0,C 180,E1 15687.118,E2 15687.118} C_VEL
LIN {X 0,Y 342.733,Z 437.55,A -85,B 0,C 180,E1 15684.794,E2 15684.794} C_VEL
LIN {X 0,Y 337.555,Z 430.155,A -85,B 0,C 180,E1 15682.647,E2 15682.647} C_VEL
LIN {X 0,Y 334.124,Z 424.137,A -85,B 0,C 180,E1 15680.311,E2 15680.311} C_VEL
LIN {X 0,Y 331.195,Z 419.145,A -85,B 0,C 180,E1 15678.116,E2 15678.116} C_VEL
LIN {X 0,Y 328.847,Z 414.988,A -85,B 0,C 180,E1 15676.118,E2 15676.118} C_VEL
LIN {X 0,Y 325.732,Z 410.191,A -85,B 0,C 180,E1 15673.309,E2 15673.309} C_VEL
LIN {X 0,Y 325.159,Z 408.886,A -85,B 0,C 180,E1 15672.61,E2 15672.61} C_VEL
LIN {X 0,Y 322.369,Z 405.077,A -85,B 0,C 180,E1 15669.641,E2 15669.641} C_VEL
LIN {X 0,Y 321.623,Z 403.265,A -85,B 0,C 180,E1 15668.401,E2 15668.401} C_VEL
LIN {X 0,Y 318.366,Z 398.528,A -85,B 0,C 180,E1 15662.88,E2 15662.88} C_VEL
LIN {X 0,Y 317.471,Z 397.182,A -85,B 0,C 180,E1 15660.36,E2 15660.36} C_VEL
LIN {X 0,Y 316.518,Z 396.34,A -85,B 0,C 180,E1 15654.743,E2 15654.743} C_VEL
LIN {X 0,Y 317.692,Z 397.341,A -85,B 0,C 180,E1 15648.931,E2 15648.931} C_VEL
LIN {X 0,Y 318.463,Z 399.159,A -85,B 0,C 180,E1 15646.38,E2 15646.38} C_VEL
LIN {X 0,Y 321.647,Z 403.532,A -85,B 0,C 180,E1 15641.138,E2 15641.138} C_VEL
LIN {X 0,Y 323.378,Z 407.243,A -85,B 0,C 180,E1 15638.523,E2 15638.523} C_VEL
LIN {X 0,Y 324.918,Z 409.132,A -85,B 0,C 180,E1 15636.994,E2 15636.994} C_VEL
LIN {X 0,Y 327.536,Z 412.787,A -85,B 0,C 180,E1 15635.374,E2 15635.374} C_VEL
LIN {X 0,Y 330.426,Z 415.479,A -85,B 0,C 180,E1 15633.974,E2 15633.974} C_VEL
LIN {X 0,Y 334.336,Z 420.048,A -85,B 0,C 180,E1 15632.19,E2 15632.19} C_VEL
LIN {X 0,Y 336.012,Z 422.061,A -85,B 0,C 180,E1 15631.471,E2 15631.471} C_VEL
LIN {X 0,Y 340.615,Z 427.508,A -85,B 0,C 180,E1 15629.626,E2 15629.626} C_VEL
LIN {X 0,Y 345.405,Z 433.439,A -85,B 0,C 180,E1 15627.865,E2 15627.865} C_VEL
LIN {X 0,Y 352.411,Z 442.237,A -85,B 0,C 180,E1 15625.526,E2 15625.526} C_VEL
LIN {X 0,Y 362.305,Z 455.925,A -85,B 0,C 180,E1 15622.567,E2 15622.567} C_VEL
LIN {X 0,Y 371.923,Z 470.458,A -85,B 0,C 180,E1 15619.995,E2 15619.995} C_VEL
LIN {X 0,Y 376.812,Z 478.723,A -85,B 0,C 180,E1 15618.768,E2 15618.768} C_VEL
LIN {X 0,Y 367.812,Z 669.597,A -85,B 0,C 180,E1 15615.057,E2 15615.057} C_VEL
LIN {X 0,Y 366.268,Z 690.168,A -85,B 0,C 180,E1 15614.396,E2 15614.396} C_VEL
LIN {X 0,Y 363.829,Z 710.88,A -85,B 0,C 180,E1 15613.46,E2 15613.46} C_VEL
LIN {X 0,Y 360.783,Z 730.015,A -85,B 0,C 180,E1 15612.327,E2 15612.327} C_VEL
LIN {X 0,Y 356.946,Z 749.077,A -85,B 0,C 180,E1 15610.896,E2 15610.896} C_VEL
LIN {X 0,Y 352.592,Z 766.981,A -85,B 0,C 180,E1 15609.22,E2 15609.22} C_VEL
LIN {X 0,Y 347.964,Z 783.63,A -85,B 0,C 180,E1 15607.317,E2 15607.317} C_VEL
LIN {X 0,Y 343.025,Z 799.597,A -85,B 0,C 180,E1 15605.106,E2 15605.106} C_VEL
LIN {X 0,Y 338.24,Z 813.774,A -85,B 0,C 180,E1 15602.745,E2 15602.745} C_VEL
LIN {X 0,Y 333.148,Z 827.863,A -85,B 0,C 180,E1 15599.877,E2 15599.877} C_VEL
LIN {X 0,Y 328.667,Z 839.62,A -85,B 0,C 180,E1 15596.951,E2 15596.951} C_VEL
LIN {X 0,Y 324.669,Z 850.027,A -85,B 0,C 180,E1 15593.79,E2 15593.79} C_VEL
LIN {X 0,Y 321.219,Z 859.077,A -85,B 0,C 180,E1 15590.4,E2 15590.4} C_VEL
LIN {X 0,Y 318.472,Z 866.713,A -85,B 0,C 180,E1 15586.786,E2 15586.786} C_VEL
LIN {X 0,Y 316.39,Z 872.845,A -85,B 0,C 180,E1 15582.964,E2 15582.964} C_VEL
LIN {X 0,Y 315.097,Z 877.187,A -85,B 0,C 180,E1 15579.127,E2 15579.127} C_VEL
LIN {X 0,Y 314.363,Z 879.964,A -85,B 0,C 180,E1 15575.291,E2 15575.291} C_VEL
LIN {X 0,Y 314.059,Z 881.291,A -85,B 0,C 180,E1 15571.276,E2 15571.276} C_VEL
LIN {X 0,Y 314.118,Z 881.098,A -85,B 0,C 180,E1 15567.446,E2 15567.446} C_VEL
LIN {X 0,Y 314.51,Z 879.438,A -85,B 0,C 180,E1 15563.612,E2 15563.612} C_VEL
LIN {X 0,Y 315.378,Z 876.208,A -85,B 0,C 180,E1 15559.774,E2 15559.774} C_VEL
LIN {X 0,Y 316.849,Z 871.381,A -85,B 0,C 180,E1 15555.938,E2 15555.938} C_VEL
LIN {X 0,Y 319.15,Z 864.786,A -85,B 0,C 180,E1 15552.121,E2 15552.121} C_VEL
LIN {X 0,Y 322.008,Z 857.095,A -85,B 0,C 180,E1 15548.674,E2 15548.674} C_VEL
LIN {X 0,Y 323.355,Z 853.579,A -85,B 0,C 180,E1 15547.336,E2 15547.336} C_VEL
LIN {X 0,Y 323.776,Z 850.444,A -85,B 0,C 180,E1 15546.08,E2 15546.08} C_VEL
LIN {X 0,Y 321.914,Z 842.43,A -85,B 0,C 180,E1 15542.823,E2 15542.823} C_VEL
LIN {X 0,Y 322.649,Z 838.529,A -85,B 0,C 180,E1 15541.632,E2 15541.632} C_VEL
LIN {X 0,Y 327.376,Z 826.518,A -85,B 0,C 180,E1 15538.724,E2 15538.724} C_VEL
LIN {X 0,Y 332.497,Z 812.858,A -85,B 0,C 180,E1 15535.994,E2 15535.994} C_VEL
LIN {X 0,Y 337.682,Z 798.128,A -85,B 0,C 180,E1 15533.567,E2 15533.567} C_VEL
LIN {X 0,Y 342.781,Z 781.939,A -85,B 0,C 180,E1 15531.379,E2 15531.379} C_VEL
LIN {X 0,Y 347.429,Z 765.412,A -85,B 0,C 180,E1 15529.541,E2 15529.541} C_VEL
LIN {X 0,Y 351.942,Z 746.939,A -85,B 0,C 180,E1 15527.859,E2 15527.859} C_VEL
LIN {X 0,Y 355.545,Z 729.464,A -85,B 0,C 180,E1 15526.566,E2 15526.566} C_VEL
LIN {X 0,Y 358.671,Z 710.067,A -85,B 0,C 180,E1 15525.434,E2 15525.434} C_VEL
LIN {X 0,Y 361.041,Z 690.051,A -85,B 0,C 180,E1 15524.545,E2 15524.545} C_VEL
LIN {X 0,Y 362.645,Z 668.5,A -85,B 0,C 180,E1 15523.869,E2 15523.869} C_VEL
LIN {X 0,Y 371.726,Z 482.088,A -85,B 0,C 180,E1 15520.197,E2 15520.197} C_VEL
LIN {X 0,Y 362.062,Z 466.738,A -85,B 0,C 180,E1 15517.612,E2 15517.612} C_VEL
LIN {X 0,Y 352.261,Z 452.683,A -85,B 0,C 180,E1 15514.688,E2 15514.688} C_VEL
LIN {X 0,Y 344.584,Z 442.605,A -85,B 0,C 180,E1 15512.123,E2 15512.123} C_VEL
LIN {X 0,Y 340.195,Z 437.103,A -85,B 0,C 180,E1 15510.513,E2 15510.513} C_VEL
LIN {X 0,Y 336.541,Z 432.55,A -85,B 0,C 180,E1 15509.062,E2 15509.062} C_VEL
LIN {X 0,Y 332.256,Z 427.386,A -85,B 0,C 180,E1 15507.221,E2 15507.221} C_VEL
LIN {X 0,Y 327.441,Z 421.775,A -85,B 0,C 180,E1 15504.923,E2 15504.923} C_VEL
LIN {X 0,Y 323.584,Z 417.647,A -85,B 0,C 180,E1 15502.865,E2 15502.865} C_VEL
LIN {X 0,Y 322.214,Z 415.947,A -85,B 0,C 180,E1 15502.054,E2 15502.054} C_VEL
LIN {X 0,Y 318.19,Z 412.047,A -85,B 0,C 180,E1 15499.457,E2 15499.457} C_VEL
LIN {X 0,Y 317.216,Z 409.89,A -85,B 0,C 180,E1 15497.993,E2 15497.993} C_VEL
LIN {X 0,Y 313.908,Z 404.461,A -85,B 0,C 180,E1 15490.832,E2 15490.832} C_VEL
LIN {X 0,Y 312.885,Z 403.545,A -85,B 0,C 180,E1 15485.134,E2 15485.134} C_VEL
LIN {X 0,Y 314.009,Z 404.485,A -85,B 0,C 180,E1 15479.271,E2 15479.271} C_VEL
LIN {X 0,Y 314.804,Z 406.468,A -85,B 0,C 180,E1 15476.541,E2 15476.541} C_VEL
LIN {X 0,Y 318.001,Z 410.576,A -85,B 0,C 180,E1 15471.502,E2 15471.502} C_VEL
LIN {X 0,Y 319.664,Z 414.221,A -85,B 0,C 180,E1 15469.001,E2 15469.001} C_VEL
LIN {X 0,Y 321.303,Z 416.076,A -85,B 0,C 180,E1 15467.419,E2 15467.419} C_VEL
LIN {X 0,Y 323.381,Z 420.104,A -85,B 0,C 180,E1 15465.13,E2 15465.13} C_VEL
LIN {X 0,Y 324.609,Z 421.885,A -85,B 0,C 180,E1 15464.09,E2 15464.09} C_VEL
LIN {X 0,Y 327.728,Z 427.281,A -85,B 0,C 180,E1 15461.501,E2 15461.501} C_VEL
LIN {X 0,Y 330.267,Z 431.004,A -85,B 0,C 180,E1 15459.996,E2 15459.996} C_VEL
LIN {X 0,Y 336.039,Z 438.755,A -85,B 0,C 180,E1 15457.429,E2 15457.429} C_VEL
LIN {X 0,Y 342.758,Z 448.095,A -85,B 0,C 180,E1 15454.793,E2 15454.793} C_VEL
LIN {X 0,Y 349.817,Z 458.322,A -85,B 0,C 180,E1 15452.325,E2 15452.325} C_VEL
LIN {X 0,Y 358.404,Z 471.69,A -85,B 0,C 180,E1 15449.626,E2 15449.626} C_VEL
LIN {X 0,Y 367.907,Z 487.764,A -85,B 0,C 180,E1 15446.936,E2 15446.936} C_VEL
LIN {X 0,Y 372.978,Z 497.439,A -85,B 0,C 180,E1 15445.577,E2 15445.577} C_VEL
LIN {X 0,Y 373.328,Z 506.489,A -85,B 0,C 180,E1 15445.218,E2 15445.218} C_VEL
LIN {X 0,Y 360.931,Z 727.603,A -85,B 0,C 180,E1 15440.608,E2 15440.608} C_VEL
LIN {X 0,Y 358.878,Z 749.882,A -85,B 0,C 180,E1 15440.005,E2 15440.005} C_VEL
LIN {X 0,Y 355.552,Z 772.298,A -85,B 0,C 180,E1 15439.175,E2 15439.175} C_VEL
LIN {X 0,Y 351.623,Z 792.849,A -85,B 0,C 180,E1 15438.154,E2 15438.154} C_VEL
LIN {X 0,Y 346.958,Z 813.922,A -85,B 0,C 180,E1 15436.805,E2 15436.805} C_VEL
LIN {X 0,Y 341.977,Z 833.906,A -85,B 0,C 180,E1 15435.201,E2 15435.201} C_VEL
LIN {X 0,Y 336.51,Z 853.736,A -85,B 0,C 180,E1 15433.221,E2 15433.221} C_VEL
LIN {X 0,Y 331.086,Z 872.221,A -85,B 0,C 180,E1 15430.977,E2 15430.977} C_VEL
LIN {X 0,Y 325.621,Z 890.306,A -85,B 0,C 180,E1 15428.332,E2 15428.332} C_VEL
LIN {X 0,Y 320.638,Z 906.787,A -85,B 0,C 180,E1 15425.448,E2 15425.448} C_VEL
LIN {X 0,Y 316.159,Z 921.795,A -85,B 0,C 180,E1 15422.305,E2 15422.305} C_VEL
LIN {X 0,Y 312.362,Z 935.461,A -85,B 0,C 180,E1 15418.902,E2 15418.902} C_VEL
LIN {X 0,Y 309.255,Z 948.134,A -85,B 0,C 180,E1 15415.141,E2 15415.141} C_VEL
LIN {X 0,Y 307.132,Z 958.7,A -85,B 0,C 180,E1 15411.382,E2 15411.382} C_VEL
LIN {X 0,Y 305.811,Z 967.527,A -85,B 0,C 180,E1 15407.504,E2 15407.504} C_VEL
LIN {X 0,Y 305.202,Z 974.889,A -85,B 0,C 180,E1 15403.449,E2 15403.449} C_VEL
LIN {X 0,Y 305.11,Z 979.932,A -85,B 0,C 180,E1 15399.811,E2 15399.811} C_VEL
LIN {X 0,Y 305.3,Z 983.341,A -85,B 0,C 180,E1 15396.204,E2 15396.204} C_VEL
LIN {X 0,Y 305.47,Z 985.219,A -85,B 0,C 180,E1 15392.815,E2 15392.815} C_VEL
LIN {X 0,Y 305.527,Z 985.672,A -85,B 0,C 180,E1 15389.438,E2 15389.438} C_VEL
LIN {X 0,Y 305.44,Z 984.812,A -85,B 0,C 180,E1 15386.247,E2 15386.247} C_VEL
LIN {X 0,Y 305.205,Z 982.459,A -85,B 0,C 180,E1 15382.661,E2 15382.661} C_VEL
LIN {X 0,Y 305.113,Z 978.467,A -85,B 0,C 180,E1 15379.045,E2 15379.045} C_VEL
LIN {X 0,Y 305.312,Z 972.667,A -85,B 0,C 180,E1 15375.203,E2 15375.203} C_VEL
LIN {X 0,Y 306.068,Z 965.481,A -85,B 0,C 180,E1 15371.528,E2 15371.528} C_VEL
LIN {X 0,Y 307.601,Z 956.088,A -85,B 0,C 180,E1 15367.65,E2 15367.65} C_VEL
LIN {X 0,Y 309.9,Z 945.377,A -85,B 0,C 180,E1 15363.977,E2 15363.977} C_VEL
LIN {X 0,Y 313.218,Z 932.322,A -85,B 0,C 180,E1 15360.259,E2 15360.259} C_VEL
LIN {X 0,Y 317.131,Z 918.388,A -85,B 0,C 180,E1 15356.95,E2 15356.95} C_VEL
LIN {X 0,Y 321.933,Z 902.286,A -85,B 0,C 180,E1 15353.73,E2 15353.73} C_VEL
LIN {X 0,Y 327.04,Z 885.657,A -85,B 0,C 180,E1 15350.945,E2 15350.945} C_VEL
LIN {X 0,Y 332.374,Z 867.829,A -85,B 0,C 180,E1 15348.453,E2 15348.453} C_VEL
LIN {X 0,Y 337.798,Z 849.012,A -85,B 0,C 180,E1 15346.286,E2 15346.286} C_VEL
LIN {X 0,Y 343.324,Z 828.428,A -85,B 0,C 180,E1 15344.342,E2 15344.342} C_VEL
LIN {X 0,Y 348.203,Z 808.387,A -85,B 0,C 180,E1 15342.813,E2 15342.813} C_VEL
LIN {X 0,Y 352.678,Z 787.406,A -85,B 0,C 180,E1 15341.551,E2 15341.551} C_VEL
LIN {X 0,Y 356.548,Z 765.751,A -85,B 0,C 180,E1 15340.57,E2 15340.57} C_VEL
LIN {X 0,Y 359.591,Z 742.682,A -85,B 0,C 180,E1 15339.791,E2 15339.791} C_VEL
LIN {X 0,Y 361.446,Z 718.141,A -85,B 0,C 180,E1 15339.192,E2 15339.192} C_VEL
LIN {X 0,Y 373.326,Z 504.739,A -85,B 0,C 180,E1 15334.754,E2 15334.754} C_VEL
LIN {X 0,Y 372.717,Z 496.781,A -85,B 0,C 180,E1 15334.38,E2 15334.38} C_VEL
LIN {X 0,Y 363.95,Z 481.009,A -85,B 0,C 180,E1 15332.02,E2 15332.02} C_VEL
LIN {X 0,Y 354.996,Z 466.364,A -85,B 0,C 180,E1 15329.391,E2 15329.391} C_VEL
LIN {X 0,Y 346.303,Z 453.191,A -85,B 0,C 180,E1 15326.538,E2 15326.538} C_VEL
LIN {X 0,Y 339.971,Z 444.268,A -85,B 0,C 180,E1 15324.221,E2 15324.221} C_VEL
LIN {X 0,Y 333.561,Z 435.489,A -85,B 0,C 180,E1 15321.589,E2 15321.589} C_VEL
LIN {X 0,Y 329.496,Z 430.178,A -85,B 0,C 180,E1 15319.73,E2 15319.73} C_VEL
LIN {X 0,Y 326.782,Z 425.647,A -85,B 0,C 180,E1 15317.816,E2 15317.816} C_VEL
LIN {X 0,Y 324.011,Z 420.775,A -85,B 0,C 180,E1 15315.389,E2 15315.389} C_VEL
LIN {X 0,Y 321.601,Z 417.002,A -85,B 0,C 180,E1 15313.118,E2 15313.118} C_VEL
LIN {X 0,Y 321.044,Z 415.694,A -85,B 0,C 180,E1 15312.409,E2 15312.409} C_VEL
LIN {X 0,Y 318.328,Z 411.85,A -85,B 0,C 180,E1 15309.4,E2 15309.4} C_VEL
LIN {X 0,Y 317.721,Z 410.239,A -85,B 0,C 180,E1 15308.323,E2 15308.323} C_VEL
LIN {X 0,Y 314.08,Z 404.615,A -85,B 0,C 180,E1 15301.459,E2 15301.459} C_VEL
LIN {X 0,Y 312.738,Z 403.457,A -85,B 0,C 180,E1 15296.333,E2 15296.333} C_VEL
LIN {X 0,Y 313.149,Z 403.789,A -85,B 0,C 180,E1 15290.999,E2 15290.999} C_VEL
LIN {X 0,Y 314.132,Z 404.897,A -85,B 0,C 180,E1 15287.873,E2 15287.873} C_VEL
LIN {X 0,Y 317.504,Z 410.404,A -85,B 0,C 180,E1 15281.263,E2 15281.263} C_VEL
LIN {X 0,Y 318.724,Z 412.788,A -85,B 0,C 180,E1 15279.909,E2 15279.909} C_VEL
LIN {X 0,Y 323.076,Z 416.897,A -85,B 0,C 180,E1 15277.241,E2 15277.241} C_VEL
LIN {X 0,Y 326.619,Z 421.098,A -85,B 0,C 180,E1 15275.3,E2 15275.3} C_VEL
LIN {X 0,Y 328.549,Z 423.017,A -85,B 0,C 180,E1 15274.348,E2 15274.348} C_VEL
LIN {X 0,Y 332.681,Z 427.767,A -85,B 0,C 180,E1 15272.429,E2 15272.429} C_VEL
LIN {X 0,Y 338.484,Z 434.967,A -85,B 0,C 180,E1 15270.003,E2 15270.003} C_VEL
LIN {X 0,Y 342.996,Z 440.629,A -85,B 0,C 180,E1 15268.302,E2 15268.302} C_VEL
LIN {X 0,Y 349.774,Z 449.338,A -85,B 0,C 180,E1 15265.975,E2 15265.975} C_VEL
LIN {X 0,Y 359.169,Z 462.529,A -85,B 0,C 180,E1 15263.086,E2 15263.086} C_VEL
LIN {X 0,Y 368.381,Z 476.699,A -85,B 0,C 180,E1 15260.545,E2 15260.545} C_VEL
LIN {X 0,Y 371.734,Z 482.466,A -85,B 0,C 180,E1 15259.669,E2 15259.669} C_VEL
LIN {X 0,Y 362.477,Z 670.346,A -85,B 0,C 180,E1 15255.984,E2 15255.984} C_VEL
LIN {X 0,Y 360.862,Z 691.119,A -85,B 0,C 180,E1 15255.313,E2 15255.313} C_VEL
LIN {X 0,Y 358.378,Z 711.529,A -85,B 0,C 180,E1 15254.387,E2 15254.387} C_VEL
LIN {X 0,Y 355.254,Z 730.606,A -85,B 0,C 180,E1 15253.255,E2 15253.255} C_VEL
LIN {X 0,Y 351.373,Z 749.242,A -85,B 0,C 180,E1 15251.852,E2 15251.852} C_VEL
LIN {X 0,Y 346.95,Z 766.957,A -85,B 0,C 180,E1 15250.2,E2 15250.2} C_VEL
LIN {X 0,Y 341.99,Z 784.286,A -85,B 0,C 180,E1 15248.221,E2 15248.221} C_VEL
LIN {X 0,Y 337.043,Z 799.786,A -85,B 0,C 180,E1 15246.071,E2 15246.071} C_VEL
LIN {X 0,Y 331.957,Z 814.265,A -85,B 0,C 180,E1 15243.652,E2 15243.652} C_VEL
LIN {X 0,Y 326.895,Z 827.676,A -85,B 0,C 180,E1 15240.917,E2 15240.917} C_VEL
LIN {X 0,Y 322.136,Z 839.697,A -85,B 0,C 180,E1 15237.945,E2 15237.945} C_VEL
LIN {X 0,Y 317.601,Z 850.95,A -85,B 0,C 180,E1 15234.519,E2 15234.519} C_VEL
LIN {X 0,Y 313.942,Z 860.066,A -85,B 0,C 180,E1 15231.066,E2 15231.066} C_VEL
LIN {X 0,Y 311.01,Z 867.74,A -85,B 0,C 180,E1 15227.394,E2 15227.394} C_VEL
LIN {X 0,Y 308.75,Z 873.918,A -85,B 0,C 180,E1 15223.481,E2 15223.481} C_VEL
LIN {X 0,Y 307.333,Z 878.342,A -85,B 0,C 180,E1 15219.549,E2 15219.549} C_VEL
LIN {X 0,Y 306.522,Z 881.196,A -85,B 0,C 180,E1 15215.615,E2 15215.615} C_VEL
LIN {X 0,Y 306.182,Z 882.582,A -85,B 0,C 180,E1 15211.683,E2 15211.683} C_VEL
LIN {X 0,Y 306.217,Z 882.536,A -85,B 0,C 180,E1 15207.754,E2 15207.754} C_VEL
LIN {X 0,Y 306.592,Z 880.963,A -85,B 0,C 180,E1 15203.822,E2 15203.822} C_VEL
LIN {X 0,Y 307.471,Z 877.905,A -85,B 0,C 180,E1 15199.887,E2 15199.887} C_VEL
LIN {X 0,Y 309.066,Z 872.99,A -85,B 0,C 180,E1 15195.768,E2 15195.768} C_VEL
LIN {X 0,Y 311.34,Z 866.861,A -85,B 0,C 180,E1 15192.044,E2 15192.044} C_VEL
LIN {X 0,Y 314.428,Z 858.979,A -85,B 0,C 180,E1 15188.356,E2 15188.356} C_VEL
LIN {X 0,Y 318.435,Z 849.048,A -85,B 0,C 180,E1 15184.723,E2 15184.723} C_VEL
LIN {X 0,Y 322.649,Z 838.529,A -85,B 0,C 180,E1 15181.632,E2 15181.632} C_VEL
LIN {X 0,Y 323.488,Z 834.54,A -85,B 0,C 180,E1 15180.459,E2 15180.459} C_VEL
LIN {X 0,Y 322.782,Z 824.504,A -85,B 0,C 180,E1 15177.37,E2 15177.37} C_VEL
LIN {X 0,Y 323.834,Z 819.826,A -85,B 0,C 180,E1 15176.287,E2 15176.287} C_VEL
LIN {X 0,Y 329.246,Z 805.437,A -85,B 0,C 180,E1 15173.692,E2 15173.692} C_VEL
LIN {X 0,Y 334.461,Z 790.401,A -85,B 0,C 180,E1 15171.446,E2 15171.446} C_VEL
LIN {X 0,Y 339.582,Z 773.75,A -85,B 0,C 180,E1 15169.409,E2 15169.409} C_VEL
LIN {X 0,Y 344.318,Z 756.192,A -85,B 0,C 180,E1 15167.651,E2 15167.651} C_VEL
LIN {X 0,Y 348.527,Z 737.784,A -85,B 0,C 180,E1 15166.151,E2 15166.151} C_VEL
LIN {X 0,Y 352.138,Z 718.454,A -85,B 0,C 180,E1 15164.898,E2 15164.898} C_VEL
LIN {X 0,Y 354.956,Z 698.552,A -85,B 0,C 180,E1 15163.902,E2 15163.902} C_VEL
LIN {X 0,Y 356.854,Z 678.517,A -85,B 0,C 180,E1 15163.173,E2 15163.173} C_VEL
LIN {X 0,Y 358.232,Z 652.013,A -85,B 0,C 180,E1 15162.534,E2 15162.534} C_VEL
LIN {X 0,Y 366.767,Z 485.968,A -85,B 0,C 180,E1 15159.278,E2 15159.278} C_VEL
LIN {X 0,Y 357.693,Z 471.548,A -85,B 0,C 180,E1 15156.741,E2 15156.741} C_VEL
LIN {X 0,Y 349.049,Z 458.998,A -85,B 0,C 180,E1 15154.057,E2 15154.057} C_VEL
LIN {X 0,Y 341.751,Z 449.262,A -85,B 0,C 180,E1 15151.532,E2 15151.532} C_VEL
LIN {X 0,Y 337.461,Z 443.787,A -85,B 0,C 180,E1 15149.902,E2 15149.902} C_VEL
LIN {X 0,Y 334.077,Z 439.527,A -85,B 0,C 180,E1 15148.514,E2 15148.514} C_VEL
LIN {X 0,Y 330.068,Z 434.607,A -85,B 0,C 180,E1 15146.734,E2 15146.734} C_VEL
LIN {X 0,Y 325.525,Z 429.212,A -85,B 0,C 180,E1 15144.498,E2 15144.498} C_VEL
LIN {X 0,Y 321.693,Z 424.925,A -85,B 0,C 180,E1 15142.38,E2 15142.38} C_VEL
LIN {X 0,Y 320.415,Z 423.449,A -85,B 0,C 180,E1 15141.606,E2 15141.606} C_VEL
LIN {X 0,Y 316.365,Z 419.268,A -85,B 0,C 180,E1 15138.902,E2 15138.902} C_VEL
LIN {X 0,Y 314.792,Z 417.396,A -85,B 0,C 180,E1 15137.676,E2 15137.676} C_VEL
LIN {X 0,Y 310.698,Z 413.502,A -85,B 0,C 180,E1 15133.587,E2 15133.587} C_VEL
LIN {X 0,Y 309.983,Z 411.394,A -85,B 0,C 180,E1 15130.595,E2 15130.595} C_VEL
LIN {X 0,Y 309.041,Z 410.562,A -85,B 0,C 180,E1 15125.012,E2 15125.012} C_VEL
LIN {X 0,Y 310.164,Z 411.507,A -85,B 0,C 180,E1 15119.262,E2 15119.262} C_VEL
LIN {X 0,Y 310.943,Z 413.569,A -85,B 0,C 180,E1 15116.498,E2 15116.498} C_VEL
LIN {X 0,Y 313.966,Z 417.616,A -85,B 0,C 180,E1 15111.577,E2 15111.577} C_VEL
LIN {X 0,Y 315.87,Z 421.405,A -85,B 0,C 180,E1 15108.867,E2 15108.867} C_VEL
LIN {X 0,Y 317.289,Z 423.273,A -85,B 0,C 180,E1 15107.442,E2 15107.442} C_VEL
LIN {X 0,Y 319.728,Z 427.279,A -85,B 0,C 180,E1 15105.142,E2 15105.142} C_VEL
LIN {X 0,Y 321.281,Z 429.421,A -85,B 0,C 180,E1 15104.152,E2 15104.152} C_VEL
LIN {X 0,Y 325.506,Z 434.885,A -85,B 0,C 180,E1 15101.788,E2 15101.788} C_VEL
LIN {X 0,Y 329.569,Z 440.318,A -85,B 0,C 180,E1 15099.766,E2 15099.766} C_VEL
LIN {X 0,Y 333.788,Z 446.001,A -85,B 0,C 180,E1 15097.872,E2 15097.872} C_VEL
LIN {X 0,Y 340.283,Z 455.242,A -85,B 0,C 180,E1 15095.247,E2 15095.247} C_VEL
LIN {X 0,Y 347.556,Z 465.956,A -85,B 0,C 180,E1 15092.641,E2 15092.641} C_VEL
LIN {X 0,Y 355.909,Z 479.399,A -85,B 0,C 180,E1 15089.95,E2 15089.95} C_VEL
LIN {X 0,Y 364.469,Z 494.311,A -85,B 0,C 180,E1 15087.45,E2 15087.45} C_VEL
LIN {X 0,Y 368.208,Z 501.621,A -85,B 0,C 180,E1 15086.408,E2 15086.408} C_VEL
LIN {X 0,Y 368.342,Z 508.039,A -85,B 0,C 180,E1 15086.168,E2 15086.168} C_VEL
LIN {X 0,Y 355.557,Z 727.533,A -85,B 0,C 180,E1 15081.56,E2 15081.56} C_VEL
LIN {X 0,Y 353.378,Z 749.806,A -85,B 0,C 180,E1 15080.944,E2 15080.944} C_VEL
LIN {X 0,Y 349.999,Z 771.808,A -85,B 0,C 180,E1 15080.122,E2 15080.122} C_VEL
LIN {X 0,Y 345.92,Z 792.315,A -85,B 0,C 180,E1 15079.094,E2 15079.094} C_VEL
LIN {X 0,Y 341.093,Z 813.26,A -85,B 0,C 180,E1 15077.739,E2 15077.739} C_VEL
LIN {X 0,Y 336.073,Z 832.655,A -85,B 0,C 180,E1 15076.171,E2 15076.171} C_VEL
LIN {X 0,Y 330.338,Z 852.591,A -85,B 0,C 180,E1 15074.165,E2 15074.165} C_VEL
LIN {X 0,Y 324.722,Z 870.878,A -85,B 0,C 180,E1 15071.922,E2 15071.922} C_VEL
LIN {X 0,Y 319.056,Z 888.793,A -85,B 0,C 180,E1 15069.27,E2 15069.27} C_VEL
LIN {X 0,Y 313.776,Z 905.294,A -85,B 0,C 180,E1 15066.345,E2 15066.345} C_VEL
LIN {X 0,Y 308.899,Z 920.789,A -85,B 0,C 180,E1 15063.035,E2 15063.035} C_VEL
LIN {X 0,Y 304.802,Z 934.704,A -85,B 0,C 180,E1 15059.473,E2 15059.473} C_VEL
LIN {X 0,Y 301.466,Z 947.512,A -85,B 0,C 180,E1 15055.539,E2 15055.539} C_VEL
LIN {X 0,Y 299.28,Z 957.773,A -85,B 0,C 180,E1 15051.758,E2 15051.758} C_VEL
LIN {X 0,Y 297.886,Z 966.529,A -85,B 0,C 180,E1 15047.784,E2 15047.784} C_VEL
LIN {X 0,Y 297.264,Z 973.507,A -85,B 0,C 180,E1 15043.816,E2 15043.816} C_VEL
LIN {X 0,Y 297.178,Z 978.571,A -85,B 0,C 180,E1 15040.076,E2 15040.076} C_VEL
LIN {X 0,Y 297.373,Z 981.997,A -85,B 0,C 180,E1 15036.37,E2 15036.37} C_VEL
LIN {X 0,Y 297.572,Z 983.809,A -85,B 0,C 180,E1 15033.082,E2 15033.082} C_VEL
LIN {X 0,Y 297.639,Z 984.369,A -85,B 0,C 180,E1 15029.616,E2 15029.616} C_VEL
LIN {X 0,Y 297.548,Z 983.561,A -85,B 0,C 180,E1 15026.34,E2 15026.34} C_VEL
LIN {X 0,Y 297.297,Z 981.395,A -85,B 0,C 180,E1 15022.805,E2 15022.805} C_VEL
LIN {X 0,Y 297.172,Z 977.344,A -85,B 0,C 180,E1 15018.945,E2 15018.945} C_VEL
LIN {X 0,Y 297.373,Z 971.627,A -85,B 0,C 180,E1 15014.998,E2 15014.998} C_VEL
LIN {X 0,Y 298.161,Z 964.48,A -85,B 0,C 180,E1 15011.223,E2 15011.223} C_VEL
LIN {X 0,Y 299.775,Z 955.176,A -85,B 0,C 180,E1 15007.241,E2 15007.241} C_VEL
LIN {X 0,Y 302.203,Z 944.562,A -85,B 0,C 180,E1 15003.474,E2 15003.474} C_VEL
LIN {X 0,Y 305.634,Z 931.783,A -85,B 0,C 180,E1 14999.729,E2 14999.729} C_VEL
LIN {X 0,Y 309.814,Z 917.745,A -85,B 0,C 180,E1 14996.287,E2 14996.287} C_VEL
LIN {X 0,Y 314.844,Z 901.776,A -85,B 0,C 180,E1 14993.006,E2 14993.006} C_VEL
LIN {X 0,Y 320.137,Z 885.431,A -85,B 0,C 180,E1 14990.194,E2 14990.194} C_VEL
LIN {X 0,Y 325.725,Z 867.565,A -85,B 0,C 180,E1 14987.646,E2 14987.646} C_VEL
LIN {X 0,Y 331.362,Z 848.953,A -85,B 0,C 180,E1 14985.455,E2 14985.455} C_VEL
LIN {X 0,Y 337.033,Z 828.813,A -85,B 0,C 180,E1 14983.509,E2 14983.509} C_VEL
LIN {X 0,Y 342.125,Z 808.919,A -85,B 0,C 180,E1 14981.953,E2 14981.953} C_VEL
LIN {X 0,Y 346.835,Z 787.669,A -85,B 0,C 180,E1 14980.655,E2 14980.655} C_VEL
LIN {X 0,Y 350.892,Z 766.041,A -85,B 0,C 180,E1 14979.654,E2 14979.654} C_VEL
LIN {X 0,Y 354.085,Z 743.145,A -85,B 0,C 180,E1 14978.862,E2 14978.862} C_VEL
LIN {X 0,Y 355.987,Z 720.137,A -85,B 0,C 180,E1 14978.281,E2 14978.281} C_VEL
LIN {X 0,Y 368.359,Z 506.014,A -85,B 0,C 180,E1 14973.798,E2 14973.798} C_VEL
LIN {X 0,Y 367.953,Z 500.934,A -85,B 0,C 180,E1 14973.548,E2 14973.548} C_VEL
LIN {X 0,Y 359.868,Z 486.267,A -85,B 0,C 180,E1 14971.279,E2 14971.279} C_VEL
LIN {X 0,Y 351.411,Z 472.185,A -85,B 0,C 180,E1 14968.694,E2 14968.694} C_VEL
LIN {X 0,Y 343.126,Z 459.417,A -85,B 0,C 180,E1 14965.872,E2 14965.872} C_VEL
LIN {X 0,Y 337.048,Z 450.707,A -85,B 0,C 180,E1 14963.561,E2 14963.561} C_VEL
LIN {X 0,Y 331.258,Z 442.613,A -85,B 0,C 180,E1 14961.096,E2 14961.096} C_VEL
LIN {X 0,Y 327.035,Z 436.999,A -85,B 0,C 180,E1 14959.095,E2 14959.095} C_VEL
LIN {X 0,Y 323.847,Z 432.785,A -85,B 0,C 180,E1 14957.426,E2 14957.426} C_VEL
LIN {X 0,Y 319.8,Z 427.398,A -85,B 0,C 180,E1 14955.04,E2 14955.04} C_VEL
LIN {X 0,Y 317.343,Z 423.446,A -85,B 0,C 180,E1 14952.741,E2 14952.741} C_VEL
LIN {X 0,Y 316.52,Z 422.118,A -85,B 0,C 180,E1 14951.848,E2 14951.848} C_VEL
LIN {X 0,Y 314.091,Z 418.019,A -85,B 0,C 180,E1 14948.789,E2 14948.789} C_VEL
LIN {X 0,Y 313.481,Z 416.946,A -85,B 0,C 180,E1 14947.883,E2 14947.883} C_VEL
LIN {X 0,Y 310.191,Z 411.566,A -85,B 0,C 180,E1 14941.292,E2 14941.292} C_VEL
LIN {X 0,Y 308.889,Z 410.469,A -85,B 0,C 180,E1 14936.102,E2 14936.102} C_VEL
LIN {X 0,Y 309.34,Z 410.843,A -85,B 0,C 180,E1 14930.699,E2 14930.699} C_VEL
LIN {X 0,Y 310.25,Z 412.016,A -85,B 0,C 180,E1 14927.719,E2 14927.719} C_VEL
LIN {X 0,Y 311.492,Z 414.606,A -85,B 0,C 180,E1 14924.929,E2 14924.929} C_VEL
LIN {X 0,Y 315.621,Z 418.22,A -85,B 0,C 180,E1 14921.435,E2 14921.435} C_VEL
LIN {X 0,Y 319.672,Z 422.875,A -85,B 0,C 180,E1 14918.63,E2 14918.63} C_VEL
LIN {X 0,Y 321.469,Z 424.601,A -85,B 0,C 180,E1 14917.555,E2 14917.555} C_VEL
LIN {X 0,Y 325.208,Z 428.947,A -85,B 0,C 180,E1 14915.476,E2 14915.476} C_VEL
LIN {X 0,Y 326.848,Z 430.783,A -85,B 0,C 180,E1 14914.642,E2 14914.642} C_VEL
LIN {X 0,Y 331.637,Z 436.528,A -85,B 0,C 180,E1 14912.384,E2 14912.384} C_VEL
LIN {X 0,Y 336.273,Z 442.28,A -85,B 0,C 180,E1 14910.424,E2 14910.424} C_VEL
LIN {X 0,Y 340.71,Z 447.955,A -85,B 0,C 180,E1 14908.706,E2 14908.706} C_VEL
LIN {X 0,Y 347.17,Z 456.437,A -85,B 0,C 180,E1 14906.429,E2 14906.429} C_VEL
LIN {X 0,Y 356.182,Z 469.318,A -85,B 0,C 180,E1 14903.579,E2 14903.579} C_VEL
LIN {X 0,Y 364.923,Z 483.031,A -85,B 0,C 180,E1 14901.091,E2 14901.091} C_VEL
LIN {X 0,Y 366.741,Z 486.388,A -85,B 0,C 180,E1 14900.592,E2 14900.592} C_VEL
LIN {X 0,Y 357.233,Z 671.201,A -85,B 0,C 180,E1 14896.937,E2 14896.937} C_VEL
LIN {X 0,Y 355.547,Z 692.087,A -85,B 0,C 180,E1 14896.257,E2 14896.257} C_VEL
LIN {X 0,Y 352.944,Z 712.684,A -85,B 0,C 180,E1 14895.315,E2 14895.315} C_VEL
LIN {X 0,Y 349.821,Z 731.187,A -85,B 0,C 180,E1 14894.212,E2 14894.212} C_VEL
LIN {X 0,Y 345.678,Z 750.397,A -85,B 0,C 180,E1 14892.757,E2 14892.757} C_VEL
LIN {X 0,Y 341.245,Z 767.557,A -85,B 0,C 180,E1 14891.147,E2 14891.147} C_VEL
LIN {X 0,Y 335.989,Z 785.297,A -85,B 0,C 180,E1 14889.11,E2 14889.11} C_VEL
LIN {X 0,Y 330.705,Z 801.212,A -85,B 0,C 180,E1 14886.875,E2 14886.875} C_VEL
LIN {X 0,Y 325.415,Z 815.677,A -85,B 0,C 180,E1 14884.422,E2 14884.422} C_VEL
LIN {X 0,Y 320.134,Z 829.065,A -85,B 0,C 180,E1 14881.644,E2 14881.644} C_VEL
LIN {X 0,Y 315.159,Z 841.068,A -85,B 0,C 180,E1 14878.62,E2 14878.62} C_VEL
LIN {X 0,Y 310.435,Z 852.225,A -85,B 0,C 180,E1 14875.157,E2 14875.157} C_VEL
LIN {X 0,Y 306.571,Z 861.365,A -85,B 0,C 180,E1 14871.623,E2 14871.623} C_VEL
LIN {X 0,Y 303.444,Z 869.085,A -85,B 0,C 180,E1 14867.842,E2 14867.842} C_VEL
LIN {X 0,Y 301.045,Z 875.26,A -85,B 0,C 180,E1 14863.833,E2 14863.833} C_VEL
LIN {X 0,Y 299.529,Z 879.678,A -85,B 0,C 180,E1 14859.8,E2 14859.8} C_VEL
LIN {X 0,Y 298.66,Z 882.527,A -85,B 0,C 180,E1 14855.763,E2 14855.763} C_VEL
LIN {X 0,Y 298.296,Z 883.91,A -85,B 0,C 180,E1 14851.728,E2 14851.728} C_VEL
LIN {X 0,Y 298.332,Z 883.864,A -85,B 0,C 180,E1 14847.695,E2 14847.695} C_VEL
LIN {X 0,Y 298.735,Z 882.294,A -85,B 0,C 180,E1 14843.659,E2 14843.659} C_VEL
LIN {X 0,Y 299.677,Z 879.24,A -85,B 0,C 180,E1 14839.621,E2 14839.621} C_VEL
LIN {X 0,Y 301.384,Z 874.33,A -85,B 0,C 180,E1 14835.397,E2 14835.397} C_VEL
LIN {X 0,Y 303.795,Z 868.208,A -85,B 0,C 180,E1 14831.583,E2 14831.583} C_VEL
LIN {X 0,Y 307.064,Z 860.331,A -85,B 0,C 180,E1 14827.809,E2 14827.809} C_VEL
LIN {X 0,Y 311.333,Z 850.285,A -85,B 0,C 180,E1 14824.058,E2 14824.058} C_VEL
LIN {X 0,Y 315.886,Z 839.465,A -85,B 0,C 180,E1 14820.83,E2 14820.83} C_VEL
LIN {X 0,Y 320.954,Z 827.111,A -85,B 0,C 180,E1 14817.814,E2 14817.814} C_VEL
LIN {X 0,Y 323.834,Z 819.826,A -85,B 0,C 180,E1 14816.287,E2 14816.287} C_VEL
LIN {X 0,Y 324.96,Z 815.041,A -85,B 0,C 180,E1 14815.228,E2 14815.228} C_VEL
LIN {X 0,Y 325.072,Z 803.063,A -85,B 0,C 180,E1 14812.375,E2 14812.375} C_VEL
LIN {X 0,Y 326.277,Z 797.642,A -85,B 0,C 180,E1 14811.422,E2 14811.422} C_VEL
LIN {X 0,Y 331.711,Z 781.565,A -85,B 0,C 180,E1 14809.267,E2 14809.267} C_VEL
LIN {X 0,Y 336.938,Z 763.953,A -85,B 0,C 180,E1 14807.34,E2 14807.34} C_VEL
LIN {X 0,Y 341.538,Z 745.664,A -85,B 0,C 180,E1 14805.721,E2 14805.721} C_VEL
LIN {X 0,Y 345.483,Z 726.705,A -85,B 0,C 180,E1 14804.375,E2 14804.375} C_VEL
LIN {X 0,Y 348.755,Z 706.503,A -85,B 0,C 180,E1 14803.252,E2 14803.252} C_VEL
LIN {X 0,Y 351.134,Z 686.218,A -85,B 0,C 180,E1 14802.411,E2 14802.411} C_VEL
LIN {X 0,Y 352.578,Z 665.128,A -85,B 0,C 180,E1 14801.81,E2 14801.81} C_VEL
LIN {X 0,Y 361.877,Z 489.892,A -85,B 0,C 180,E1 14798.328,E2 14798.328} C_VEL
LIN {X 0,Y 353.646,Z 476.718,A -85,B 0,C 180,E1 14795.921,E2 14795.921} C_VEL
LIN {X 0,Y 345.66,Z 464.998,A -85,B 0,C 180,E1 14793.34,E2 14793.34} C_VEL
LIN {X 0,Y 338.957,Z 455.907,A -85,B 0,C 180,E1 14790.931,E2 14790.931} C_VEL
LIN {X 0,Y 332.589,Z 447.512,A -85,B 0,C 180,E1 14788.359,E2 14788.359} C_VEL
LIN {X 0,Y 327.906,Z 441.82,A -85,B 0,C 180,E1 14786.241,E2 14786.241} C_VEL
LIN {X 0,Y 323.628,Z 436.642,A -85,B 0,C 180,E1 14784.068,E2 14784.068} C_VEL
LIN {X 0,Y 319.757,Z 432.096,A -85,B 0,C 180,E1 14781.846,E2 14781.846} C_VEL
LIN {X 0,Y 314.497,Z 426.337,A -85,B 0,C 180,E1 14778.25,E2 14778.25} C_VEL
LIN {X 0,Y 313.05,Z 424.891,A -85,B 0,C 180,E1 14777.089,E2 14777.089} C_VEL
LIN {X 0,Y 307.303,Z 418.961,A -85,B 0,C 180,E1 14770.688,E2 14770.688} C_VEL
LIN {X 0,Y 305.227,Z 417.598,A -85,B 0,C 180,E1 14765.263,E2 14765.263} C_VEL
LIN {X 0,Y 306.26,Z 418.466,A -85,B 0,C 180,E1 14759.439,E2 14759.439} C_VEL
LIN {X 0,Y 307.01,Z 420.358,A -85,B 0,C 180,E1 14756.827,E2 14756.827} C_VEL
LIN {X 0,Y 310.35,Z 424.742,A -85,B 0,C 180,E1 14751.758,E2 14751.758} C_VEL
LIN {X 0,Y 313.416,Z 429.104,A -85,B 0,C 180,E1 14748.872,E2 14748.872} C_VEL
LIN {X 0,Y 314.896,Z 430.803,A -85,B 0,C 180,E1 14747.718,E2 14747.718} C_VEL
LIN {X 0,Y 319.153,Z 436.314,A -85,B 0,C 180,E1 14744.789,E2 14744.789} C_VEL
LIN {X 0,Y 323.768,Z 442.569,A -85,B 0,C 180,E1 14742.105,E2 14742.105} C_VEL
LIN {X 0,Y 327.679,Z 447.924,A -85,B 0,C 180,E1 14740.11,E2 14740.11} C_VEL
LIN {X 0,Y 331.648,Z 453.378,A -85,B 0,C 180,E1 14738.281,E2 14738.281} C_VEL
LIN {X 0,Y 338.03,Z 462.677,A -85,B 0,C 180,E1 14735.63,E2 14735.63} C_VEL
LIN {X 0,Y 344.865,Z 473.01,A -85,B 0,C 180,E1 14733.11,E2 14733.11} C_VEL
LIN {X 0,Y 352.966,Z 486.314,A -85,B 0,C 180,E1 14730.423,E2 14730.423} C_VEL
LIN {X 0,Y 361.182,Z 501.072,A -85,B 0,C 180,E1 14727.94,E2 14727.94} C_VEL
LIN {X 0,Y 363.517,Z 505.802,A -85,B 0,C 180,E1 14727.261,E2 14727.261} C_VEL
LIN {X 0,Y 363.152,Z 514.591,A -85,B 0,C 180,E1 14727.04,E2 14727.04} C_VEL
LIN {X 0,Y 350.202,Z 728.573,A -85,B 0,C 180,E1 14722.515,E2 14722.515} C_VEL
LIN {X 0,Y 347.643,Z 752.111,A -85,B 0,C 180,E1 14721.831,E2 14721.831} C_VEL
LIN {X 0,Y 344.129,Z 773.445,A -85,B 0,C 180,E1 14721,E2 14721} C_VEL
LIN {X 0,Y 340.033,Z 793.1,A -85,B 0,C 180,E1 14719.99,E2 14719.99} C_VEL
LIN {X 0,Y 335.17,Z 813.187,A -85,B 0,C 180,E1 14718.661,E2 14718.661} C_VEL
LIN {X 0,Y 329.87,Z 832.734,A -85,B 0,C 180,E1 14717.049,E2 14717.049} C_VEL
LIN {X 0,Y 323.936,Z 852.552,A -85,B 0,C 180,E1 14715.023,E2 14715.023} C_VEL
LIN {X 0,Y 318.103,Z 870.624,A -85,B 0,C 180,E1 14712.756,E2 14712.756} C_VEL
LIN {X 0,Y 312.176,Z 888.458,A -85,B 0,C 180,E1 14710.05,E2 14710.05} C_VEL
LIN {X 0,Y 306.68,Z 904.723,A -85,B 0,C 180,E1 14707.092,E2 14707.092} C_VEL
LIN {X 0,Y 301.467,Z 920.517,A -85,B 0,C 180,E1 14703.63,E2 14703.63} C_VEL
LIN {X 0,Y 297.272,Z 933.948,A -85,B 0,C 180,E1 14700.074,E2 14700.074} C_VEL
LIN {X 0,Y 293.906,Z 946.072,A -85,B 0,C 180,E1 14696.246,E2 14696.246} C_VEL
LIN {X 0,Y 291.544,Z 956.336,A -85,B 0,C 180,E1 14692.374,E2 14692.374} C_VEL
LIN {X 0,Y 290.023,Z 965.124,A -85,B 0,C 180,E1 14688.283,E2 14688.283} C_VEL
LIN {X 0,Y 289.324,Z 972.123,A -85,B 0,C 180,E1 14684.203,E2 14684.203} C_VEL
LIN {X 0,Y 289.237,Z 977.209,A -85,B 0,C 180,E1 14680.355,E2 14680.355} C_VEL
LIN {X 0,Y 289.44,Z 980.652,A -85,B 0,C 180,E1 14676.546,E2 14676.546} C_VEL
LIN {X 0,Y 289.674,Z 982.477,A -85,B 0,C 180,E1 14673.166,E2 14673.166} C_VEL
LIN {X 0,Y 289.75,Z 983.041,A -85,B 0,C 180,E1 14669.605,E2 14669.605} C_VEL
LIN {X 0,Y 289.643,Z 982.227,A -85,B 0,C 180,E1 14666.24,E2 14666.24} C_VEL
LIN {X 0,Y 289.375,Z 980.084,A -85,B 0,C 180,E1 14662.656,E2 14662.656} C_VEL
LIN {X 0,Y 289.231,Z 976.221,A -85,B 0,C 180,E1 14658.84,E2 14658.84} C_VEL
LIN {X 0,Y 289.437,Z 970.587,A -85,B 0,C 180,E1 14654.781,E2 14654.781} C_VEL
LIN {X 0,Y 290.328,Z 963.013,A -85,B 0,C 180,E1 14650.668,E2 14650.668} C_VEL
LIN {X 0,Y 292.105,Z 953.576,A -85,B 0,C 180,E1 14646.54,E2 14646.54} C_VEL
LIN {X 0,Y 294.852,Z 942.468,A -85,B 0,C 180,E1 14642.54,E2 14642.54} C_VEL
LIN {X 0,Y 298.718,Z 929.205,A -85,B 0,C 180,E1 14638.597,E2 14638.597} C_VEL
LIN {X 0,Y 303.365,Z 914.576,A -85,B 0,C 180,E1 14635.011,E2 14635.011} C_VEL
LIN {X 0,Y 308.654,Z 898.774,A -85,B 0,C 180,E1 14631.782,E2 14631.782} C_VEL
LIN {X 0,Y 314.472,Z 881.523,A -85,B 0,C 180,E1 14628.847,E2 14628.847} C_VEL
LIN {X 0,Y 320.236,Z 864.07,A -85,B 0,C 180,E1 14626.375,E2 14626.375} C_VEL
LIN {X 0,Y 326.185,Z 845.046,A -85,B 0,C 180,E1 14624.176,E2 14624.176} C_VEL
LIN {X 0,Y 331.917,Z 825.141,A -85,B 0,C 180,E1 14622.297,E2 14622.297} C_VEL
LIN {X 0,Y 337.199,Z 804.823,A -85,B 0,C 180,E1 14620.754,E2 14620.754} C_VEL
LIN {X 0,Y 342.03,Z 783.673,A -85,B 0,C 180,E1 14619.496,E2 14619.496} C_VEL
LIN {X 0,Y 346.141,Z 761.675,A -85,B 0,C 180,E1 14618.523,E2 14618.523} C_VEL
LIN {X 0,Y 349.112,Z 739.56,A -85,B 0,C 180,E1 14617.787,E2 14617.787} C_VEL
LIN {X 0,Y 351.235,Z 711.613,A -85,B 0,C 180,E1 14617.116,E2 14617.116} C_VEL
LIN {X 0,Y 363.49,Z 507.172,A -85,B 0,C 180,E1 14612.812,E2 14612.812} C_VEL
LIN {X 0,Y 363.214,Z 504.933,A -85,B 0,C 180,E1 14612.676,E2 14612.676} C_VEL
LIN {X 0,Y 354.337,Z 488.82,A -85,B 0,C 180,E1 14610.057,E2 14610.057} C_VEL
LIN {X 0,Y 346.463,Z 475.675,A -85,B 0,C 180,E1 14607.499,E2 14607.499} C_VEL
LIN {X 0,Y 339.091,Z 464.248,A -85,B 0,C 180,E1 14604.846,E2 14604.846} C_VEL
LIN {X 0,Y 331.938,Z 453.873,A -85,B 0,C 180,E1 14601.932,E2 14601.932} C_VEL
LIN {X 0,Y 328.277,Z 448.836,A -85,B 0,C 180,E1 14600.27,E2 14600.27} C_VEL
LIN {X 0,Y 324.778,Z 444.019,A -85,B 0,C 180,E1 14598.533,E2 14598.533} C_VEL
LIN {X 0,Y 321.751,Z 439.972,A -85,B 0,C 180,E1 14596.891,E2 14596.891} C_VEL
LIN {X 0,Y 317.954,Z 434.786,A -85,B 0,C 180,E1 14594.57,E2 14594.57} C_VEL
LIN {X 0,Y 313.896,Z 429.611,A -85,B 0,C 180,E1 14591.669,E2 14591.669} C_VEL
LIN {X 0,Y 310.471,Z 425.136,A -85,B 0,C 180,E1 14588.612,E2 14588.612} C_VEL
LIN {X 0,Y 309.719,Z 423.989,A -85,B 0,C 180,E1 14587.792,E2 14587.792} C_VEL
LIN {X 0,Y 306.33,Z 418.531,A -85,B 0,C 180,E1 14581.122,E2 14581.122} C_VEL
LIN {X 0,Y 305.045,Z 417.453,A -85,B 0,C 180,E1 14575.488,E2 14575.488} C_VEL
LIN {X 0,Y 305.893,Z 418.027,A -85,B 0,C 180,E1 14571.352,E2 14571.352} C_VEL
LIN {X 0,Y 307.901,Z 419.534,A -85,B 0,C 180,E1 14568.004,E2 14568.004} C_VEL
LIN {X 0,Y 314.21,Z 425.95,A -85,B 0,C 180,E1 14561.733,E2 14561.733} C_VEL
LIN {X 0,Y 318.325,Z 430.695,A -85,B 0,C 180,E1 14558.825,E2 14558.825} C_VEL
LIN {X 0,Y 319.803,Z 432.207,A -85,B 0,C 180,E1 14557.916,E2 14557.916} C_VEL
LIN {X 0,Y 323.637,Z 436.653,A -85,B 0,C 180,E1 14555.738,E2 14555.738} C_VEL
LIN {X 0,Y 329.533,Z 443.822,A -85,B 0,C 180,E1 14552.829,E2 14552.829} C_VEL
LIN {X 0,Y 334.176,Z 449.716,A -85,B 0,C 180,E1 14550.81,E2 14550.81} C_VEL
LIN {X 0,Y 340.63,Z 458.022,A -85,B 0,C 180,E1 14548.303,E2 14548.303} C_VEL
LIN {X 0,Y 349.622,Z 470.668,A -85,B 0,C 180,E1 14545.212,E2 14545.212} C_VEL
LIN {X 0,Y 358.743,Z 484.789,A -85,B 0,C 180,E1 14542.433,E2 14542.433} C_VEL
LIN {X 0,Y 361.852,Z 490.211,A -85,B 0,C 180,E1 14541.541,E2 14541.541} C_VEL
LIN {X 0,Y 352.101,Z 671.841,A -85,B 0,C 180,E1 14537.923,E2 14537.923} C_VEL
LIN {X 0,Y 350.342,Z 692.964,A -85,B 0,C 180,E1 14537.233,E2 14537.233} C_VEL
LIN {X 0,Y 347.723,Z 713.111,A -85,B 0,C 180,E1 14536.31,E2 14536.31} C_VEL
LIN {X 0,Y 344.486,Z 731.737,A -85,B 0,C 180,E1 14535.2,E2 14535.2} C_VEL
LIN {X 0,Y 340.308,Z 750.538,A -85,B 0,C 180,E1 14533.776,E2 14533.776} C_VEL
LIN {X 0,Y 335.551,Z 768.453,A -85,B 0,C 180,E1 14532.095,E2 14532.095} C_VEL
LIN {X 0,Y 330.169,Z 786.012,A -85,B 0,C 180,E1 14530.069,E2 14530.069} C_VEL
LIN {X 0,Y 324.831,Z 801.584,A -85,B 0,C 180,E1 14527.88,E2 14527.88} C_VEL
LIN {X 0,Y 319.294,Z 816.133,A -85,B 0,C 180,E1 14525.398,E2 14525.398} C_VEL
LIN {X 0,Y 313.747,Z 829.663,A -85,B 0,C 180,E1 14522.582,E2 14522.582} C_VEL
LIN {X 0,Y 308.514,Z 841.789,A -85,B 0,C 180,E1 14519.509,E2 14519.509} C_VEL
LIN {X 0,Y 303.757,Z 852.532,A -85,B 0,C 180,E1 14516.169,E2 14516.169} C_VEL
LIN {X 0,Y 299.606,Z 861.881,A -85,B 0,C 180,E1 14512.565,E2 14512.565} C_VEL
LIN {X 0,Y 296.039,Z 870.085,A -85,B 0,C 180,E1 14508.508,E2 14508.508} C_VEL
LIN {X 0,Y 293.448,Z 876.332,A -85,B 0,C 180,E1 14504.4,E2 14504.4} C_VEL
LIN {X 0,Y 291.79,Z 880.832,A -85,B 0,C 180,E1 14500.262,E2 14500.262} C_VEL
LIN {X 0,Y 290.799,Z 883.859,A -85,B 0,C 180,E1 14495.919,E2 14495.919} C_VEL
